IF VAT.bAbisoliererLINKSundAUF AND NOT VAT.bNurAbisolieren THEN
	VAT.bAbisoliererLINKSundAUF := FALSE;
	VAT.bCrimpeinheitVOR := TRUE; //M20.4
	GVL.EinzelschrittIdx := einzelSchrittOffset + 25; //NBT-NEU: Crimpeinheit vor
	MAIN.M_Log(reqLevel:=CVL.TRACE, objectName:= 'Ablauf', sMsg:= '4---Crimper vor',errNo := 16#FFFFFFFF);
	RETURN;
END_IF

(*	
	//*** 5---Crimpen zu
	U "M 20.4" M20.4 -- 4---Crimpeinheit vor
	R "M 20.4" M20.4 -- 4---Crimpeinheit vor
	S "M 20.5" M20.5 -- 5---Crimpen zu
	R "M 23.3" M23.3 -- S&R 2ter Vereinzelungs-Versuch
	SPB end
*)
	
IF VAT.bCrimpeinheitVOR THEN //M20.4
	VAT.bCrimpeinheitVOR := FALSE; //M20.4
	VAT.bCrimpenZU := TRUE; //M20.5
	VAT.bSr2terVereinzVersuch := FALSE; //M23.3
	GVL.EinzelschrittIdx := einzelSchrittOffset + 26; //NBT-NEU: Crimpen zu
	MAIN.M_Log(reqLevel:=CVL.TRACE, objectName:= 'Ablauf', sMsg:= '5---Crimper zu',errNo := 16#FFFFFFFF);
	RETURN;
END_IF
	
(*	
	//*** 6---Drahthalter + Drahtführung auf
	U "M 20.5" M20.5 -- 5---Crimpen zu
	R "M 20.5" M20.5 -- 5---Crimpen zu
	S "M 20.6" M20.6 -- 6---Drahthalter + Drahtführung auf
	SPB end
*)
	
IF VAT.bCrimpenZU THEN //Crimpen zu
	VAT.bCrimpenZU := FALSE;
	VAT.bDrahtHalterUndFuehrungAUF := TRUE;
	GVL.EinzelschrittIdx := einzelSchrittOffset + 27; //NBT-NEU: Drahthalter + Drahtführung auf
	MAIN.M_Log(reqLevel:=CVL.TRACE, objectName:= 'Ablauf', sMsg:= '6---Draht auf',errNo := 16#FFFFFFFF);
	RETURN;
END_IF
	
(*		
	//*** 7---Crimpzange auf + Abisoliereinheit vor
	U "M 20.6" M20.6 -- 6---Drahthalter + Drahtführung auf
	R "M 20.6" M20.6 -- 6---Drahthalter + Drahtführung auf
	S "M 20.7" M20.7 -- 7---Crimpzange auf + Abisoliereinheit vor
	SPB end
*)
		
IF VAT.bDrahtHalterUndFuehrungAUF THEN //Drahthalter + Drahtführung auf
	VAT.bDrahtHalterUndFuehrungAUF := FALSE; //M20.6
	VAT.bCrZangeAUF_AisolierVOR := TRUE; //M20.7
	GVL.EinzelschrittIdx := einzelSchrittOffset + 28; //NBT-NEU: Crimpzange auf + Abisoliereinheit vor
	MAIN.M_Log(reqLevel:=CVL.TRACE, objectName:= 'Ablauf', sMsg:= '7---C-Zange auf, AbIso vor',errNo := 16#FFFFFFFF);
	RETURN;
END_IF

(*		
	//*** 8---Ausstoßen vor
	L "DB6".w134_Ausstossverz DB6.DBW134 -- Ausstoß-Verzögerung
	L 10
	*I -- AKKU1 und AKKU2 multiplizieren, Das Ergebnis wird in AKKU 1 abgelegt.
	ITB -- Ganzzahl in BCD umwandeln (3 Stellen und eine Stelle Vorzeichen)
	
	U "M 20.7" M20.7 -- 7---Crimpzange auf + Abisoliereinheit vor
	SE "T 22" T22 -- Ausstoß-Verzögerung
	U "T 22" T22 -- Ausstoß-Verzögerung
	R "M 20.7" M20.7 -- 7 Crimpzange auf + Abisoliereinheit vor
	S "M 21.0" M21.0 -- 8---Ausstoßen vor
	SPB end
*)

//ITB ??? Wert befindet sich in AKKU 1, wird aber nicht weggeschrieben...was passiert damit?
//nach vorn verlagert
//GVL.tonAusstoss(IN := VAT.bCrZangeAUF_AisolierVOR, PT := INT_TO_TIME (nTmp)); 

IF GVL.tonAusstoss.Q THEN
	VAT.bCrZangeAUF_AisolierVOR := FALSE; //M20.7
	VAT.bAusstossenVOR := TRUE; //M21.0
	GVL.EinzelschrittIdx := einzelSchrittOffset + 29; //NBT-NEU: Ausstoßen vor
	MAIN.M_Log(reqLevel:=CVL.TRACE, objectName:= 'Ablauf', sMsg:= '8---Ausstoßen vor',errNo := 16#FFFFFFFF);
	RETURN;
ELSE	
	GVL.EinzelschrittIdx := einzelSchrittOffset + 29; //NBT-NEU: Ausstoßen vor
END_IF

(*		
	//*** 9---Crimpeinheit rück
	U "M 21.0" M21.0 -- 8---Ausstoßen vor
	R "M 21.0" M21.0 -- 8---Ausstoßen vor
	S "M 21.1" M21.1 -- 9---Crimpeinheit rück
	SPB end
*)
	
IF VAT.bAusstossenVOR THEN //M21.0
	VAT.bAusstossenVOR := FALSE;
	VAT.bCrimpeinheitRUECK := TRUE; //M21.1
	GVL.EinzelschrittIdx := einzelSchrittOffset + 30; //NBT-NEU: Crimpeinheit rück
	MAIN.M_Log(reqLevel:=CVL.TRACE, objectName:= 'Ablauf', sMsg:= '9---Crimper rück',errNo := 16#FFFFFFFF);
	RETURN;
END_IF
(*		
	//*** 10--Abisolierer nach rechts + Kontakt-Schieben rück
	U "M 20.3" M20.3 -- 3---Abisolierer nach links + Abisolierer auf
	U "M8.4NurAbisolieren" M8.4 -- Nur Abisolieren
	UN "T 20" T20 -- Ablauf-Verz.bei Probelauf
	O "M 21.1" M21.1 -- 9---Crimpeinheit rück
	SPBN l10
*)
	
//SPBN -> Springe wenn VKE = 0 -> 'Springe bei FALSE' heißt 'Tu was bei TRUE'.
IF VAT.bAbisoliererLINKSundAUF AND VAT.bNurAbisolieren AND NOT GVL.tofAblVerzProbelauf.Q OR VAT.bCrimpeinheitRUECK THEN
	
	MAIN.M_Log(reqLevel:=CVL.TRACE, objectName:= 'Ablauf', sMsg:= '10--Abisolierer re + K-Schieber rück',errNo := 16#FFFFFFFF);
	(*	
		R "M 20.3" M20.3 -- 3---Abisolierer nach links + Abisolierer auf
		R "M 21.1" M21.1 -- 9---Crimpeinheit rück
		S "M 21.2" M21.2 -- 10--Abisolierer nach rechts + Kontakt-Schieben rück
	*)
	VAT.bAbisoliererLINKSundAUF := FALSE; //M20.3
	VAT.bCrimpeinheitRUECK := FALSE; //M21.1
	VAT.bAbisoNachRE_KontSchiebRUECK := TRUE; //M21.2

	(*	
		U "M8.7ohneLitze" M8.7 -- Probelauf ohne Litze
		R "M8.7ohneLitze" M8.7 -- Probelauf ohne Litze
		R "M0.6" M0.6 -- SR Start
	*)
	
	IF VAT.bProbelOhneLitze THEN // Probelauf ohne Litze //M8.7
		VAT.bProbelOhneLitze := FALSE; //M8.7
		VAT.bSrStart := FALSE; //SR Start - M0.6
	END_IF
	
	(*	
		O "M8.5ohneKontakt" M8.5 -- Probelauf ohne Kontakt
		O "M8.6ohneCrmpen" M8.6 -- Probelauf ohne Crimpen
		L S5T#600MS
		SA "T 20" T20 -- Ablauf-Verz.bei Probelauf
		CLR
		SA "T 20" T20 -- Ablauf-Verz.bei Probelauf
	*)
	

	GVL.tofAblVerzProbelauf(IN := VAT.bProbelOhneKontakt OR VAT.bProbelOhneCrimpen, PT := T#600MS); //T20
	
	(*
		U "M8.0NormalCrimp" M8.0 -- Normal Crimpen
		SPBN l10
	*)
	
	//SPBN -> Springe wenn VKE = 0 -> 'Springe bei FALSE' heißt 'Tu was bei TRUE'.
	IF VAT.bNormalCrimp THEN // Normal Crimpen
		(*	
			L "DB6".d140_Total_Z DB6.DBD140 -- Total-Zähler
			+ L#1
			T "DB6".d140_Total_Z DB6.DBD140 -- Total-Zähler
			L "DB6".d144_Tages_Z DB6.DBD144 -- Tages-Zähler
			+ L#1
			T "DB6".d144_Tages_Z DB6.DBD144 -- Tages-Zähler
			L "DB6".d68Stueck_Fertig DB6.DBD68 -- Fertig Stückz
			+ L#1
			T "DB6".d68Stueck_Fertig DB6.DBD68 -- Fertig Stückz
			L "DB6".d64Stueck_Vorwahl DB6.DBD64 -- Stückzahl-Vorwahl Stückz
			==D
			S "A70" M107.0 -- Stückzahl-Vorwahl erreicht
			
			L "DB6".d152_WartZ_Z DB6.DBD152 -- Zähler Wartung
			+ L#1
			T "DB6".d152_WartZ_Z DB6.DBD152 -- Zähler Wartung
			
			L "DB6".d148_WartZ_V DB6.DBD148 -- Vorwahl Wartung
			==D
			S "A67" M106.7 -- Wartungs-Zähler, hat Vorwahl erreicht, weiter mit Reset
			SPA end
		*)
					
		
		DB6.diTotalZaehler := DB6.diTotalZaehler + 1;
		
		DB6.diTagesZaehler := DB6.diTagesZaehler + 1;
					
		DB6.diStueck_Fertig := DB6.diStueck_Fertig + 1;
		
		IF DB6.diStueck_Fertig = DB6.diStueck_Vorwahl THEN
			GVL.errs.StueckZaehlErreicht := TRUE; //M107.0
		END_IF
		
		
		DB6.diWartungsZaehler := DB6.diWartungsZaehler + 1;
		
		IF DB6.diWartungsZaehler = DB6.diWartZaehlVorwahl THEN
			GVL.errs.WartungsZaehlErreicht := TRUE; //M106.7
			GVL.EinzelschrittIdx := einzelSchrittOffset + 31; //NBT-NEU: Abisolierer nach rechts + Kontakt-Schieben rück
			RETURN; //Wartungs-Zähler, hat Vorwahl erreicht, weiter mit Reset
		END_IF

	END_IF // end of IF VAT.M8.0...

END_IF //end of IF VAT.M20.3 AND VAT.M8.4 AND NOT ...

(*	
l10: BLD 130
	U "M 21.2" M21.2 -- 10--Abisolierer nach rechts + Kontakt-Schieben rück
	R "M 21.2" M21.2 -- 10--Abisolierer nach rechts + Kontakt-Schieben rück
*)

IF VAT.bAbisoNachRE_KontSchiebRUECK THEN //M21.2
	VAT.bAbisoNachRE_KontSchiebRUECK := FALSE; //M21.2
	GVL.EinzelschrittIdx := einzelSchrittOffset + 32; // Einzelschritt Ende
	MAIN.M_Log(reqLevel:=CVL.TRACE, objectName:= 'Ablauf', sMsg:= '10--ENDE',errNo := 16#FFFFFFFF);
END_IF

(*	
end: BLD 130
*)

END_FUNCTION_BLOCK

// ---- POUs/MainPous/F20_Ablauf/P_AblaufReset.TcPOU
PROGRAM P_AblaufReset 
VAR
//rTrig : R_TRIG;
//bTmp:BOOL := FALSE;
tsv1 : TSV;	

END_VAR

(* Netzwerk: 2 Ablauf-Reset *)

(* 
U "E0_0" E0.0	-- Taste Start
U "M0.7" M0.7	-- Störung aufgetreten (gesammelt)
L S5T#1S		-- mandatory!
SE "T 1" T1 -- Verz. Taste Start, SE <Zeit> startet die adressierte Zeit, wenn das VKE von "0" auf "1" wechselt.
*)

(*
Klassisches TON-Verhalten:
Die programmierte Zeitdauer läuft ab, solange das VKE = 1 ist. Wechselt das VKE auf "0", bevor die programmierte
Zeitdauer abgelaufen ist, wird die Zeit angehalten. Für diese Operation (Starten der Zeit) müssen der
Zeitwert und die Zeitbasis im BCD-Format in AKKU1-L gespeichert sein.
*)
//Also nur wenn eine Sammelstörung aufgetreten ist und 1 sek. gedrückt wird!...
GVL.tonTasteStartOnErr(IN := GVL.insecTasterStart AND VAT.bSammelStoerung, PT := T#1S);

(*
	ON "T 72" T72 -- Verz. Alles OK von PNOZ
	O "T 1" T1 -- Verz. Taste Start
	SPBN res -- Springe nach 'res' wenn VKE = 0

	R "M8.1MagLeerf" M8.1 -- Magazin Leerfahren
	R "M8.2SortLeerf" M8.2 -- Sortierer Leerfahren
	R "M8.3CrimpEinr" M8.3 -- Crimpen Einrichten
	R "M8.5ohneKontakt" M8.5 -- Probelauf ohne Kontakt
	R "M8.6ohneCrmpen" M8.6 -- Probelauf ohne Crimpen
	R "M8.7ohneLitze" M8.7 -- Probelauf ohne Litze

	L 0
	T MD 20 -- Bedeutung noch Unklar
	T MW 0 -- Bedeutung noch Unklar
	T AW 0 -- Bedeutung noch Unklar
	T AW 2 -- Bedeutung noch Unklar
	T MD 104 -- Bedeutung noch Unklar
	T MD 108 -- Bedeutung noch Unklar
	SET -- 	VKE auf 1 setzen (=1)
	S "M1.3_Stop" M1.3 -- RS Stop StST
*)

IF (* NOT GVL.tonSAFETYok.Q OR *) GVL.tonTasteStartOnErr.Q THEN
	VAT.bMagazinLeerfahren := FALSE;
	VAT.bSortiererLeerfahren := FALSE;
	VAT.bCrimpEinrichten := FALSE;
	VAT.bProbelOhneKontakt := FALSE;
	VAT.bProbelOhneCrimpen := FALSE;
	VAT.bProbelOhneLitze := FALSE;
	
	//GVL.MD20 := 0; //Bedeutung noch Unklar
	//GVL.MW0 := 0; //Bedeutung noch Unklar
	//T AW 0 -- Bedeutung noch Unklar(evtl. alle 8 Ausg. auf 0)
	//T AW 2 -- Bedeutung noch Unklar (evtl. alle 8 Ausg. als WORD auf 2)
	//GVL.MD104 := 0; //war Fehererkennung, jtzt GVL.errs
	//GVL.MD108 := 0; //war Fehererkennung, jtzt GVL.errs
	
	F_ResetErrors(); //Reset Fehlerflags
	
	VAT.bRsStop := TRUE; //(ehemals M1.3) RS Stop
END_IF

(*	
res: BLD 130
	U "T 72" T72 -- Verz. Alles OK von PNOZ
	L S5T#500MS
	SV "T 19" T19 -- Kontaktauswurf nach Einschalten, Zeit als Zeit mit verlängertem Impuls starten: TSV.
*)

GVL.tsvKontauswurf(IN := GVL.tonSAFETYok.Q, PT := T#500MS);

END_PROGRAM

// ---- POUs/MainPous/FC3_FehlerAllg/F_ResetErrors.TcPOU
FUNCTION F_ResetErrors : BOOL
VAR_INPUT
END_VAR
VAR
END_VAR

//M104.0
	GVL.errs.DrahthltNichtOffen := FALSE; //(ehem. M104.0) Drahthalter nicht offen
	GVL.errs.DrahthltNichtZu := FALSE; //(ehem. M104.1) Drahthalter nicht zu
	GVL.errs.AusloesSchaltDauerMldg := FALSE;//(ehem. M104.2) -- Auslöseschalter Dauermelung
	GVL.errs.AbisolierNichtOffen  := FALSE; //(ehem. M104.3) Abisolierer nicht offen
	GVL.errs.AbisolierNichtZu  := FALSE; //(ehem. M104.4) Abisolierer nicht zu
	GVL.errs.DoppelMlgAbisoVornRueck  := FALSE; //(ehem. M104.5) Doppelmeldung Abisolierer vorn+rück
	GVL.errs.AbisolierNichtVorn  := FALSE; //(ehem. M104.6) Abisolierer nicht vorn
	GVL.errs.AbisolierNichtRueck  := FALSE; //(ehem. M104.7) Abisolierer nicht rück (abisoliert)
	
	//M105.0
	GVL.errs.AbisolierNichtLinks  := FALSE; //(ehem. M105.0) Abisolierer nicht links (aus Arbeitsraum)
	GVL.errs.AbisolierNichtRechts  := FALSE; //(ehem. M105.1) Abisolierer nicht rechts
	GVL.errs.DoppelMlgCrimpzZuOffen  := FALSE; //(ehem. M105.2) Doppelmeldung Crimpzange zu+offen
	GVL.errs.CrimpZangeNichtZu  := FALSE; //(ehem. M105.3) Crimpzange nicht zu
	GVL.errs.CrimpZangeNichtOffen  := FALSE; //(ehem. M105.4) Crimpzange nicht offen
	GVL.errs.KontaktNichtGefallen  := FALSE; //Reserve, war in AWL nicht belegt
	GVL.errs.DauerMlgKontaktGefallen  := FALSE; //Reserve, war in AWL nicht belegt
	GVL.errs.DoppelMlgCrimpEinhVornZurueck  := FALSE; //(ehem. M105.7) Doppelmeldung Crimpeinheit vorn+rück
	
	//M106.0
	GVL.errs.CrimpeinheitNichtVorn  := FALSE; //(ehem. M106.0)Crimpeinheit nicht vorn
	GVL.errs.CrimpeinheitNichtRueck  := FALSE; //(ehem. M106.1) Crimpeinheit nicht rück
	GVL.errs.KontaktSchiebenNichtVorn  := FALSE; //(ehem. M106.2) Kontakt-Schieben nicht vorn
	GVL.errs.KontaktSchiebenNichtRueck  := FALSE; //(ehem. M106.3) Kontakt-Schieben nicht rück
	GVL.errs.AusstossenNichtVorn  := FALSE; //(ehem. M106.4) Ausstoßen nicht vorn
	GVL.errs.AusstossenNichtRueck  := FALSE; //(ehem. M106.5) Ausstoßen nicht rück
	GVL.errs.r106_6  := FALSE; //Reserve, war in AWL nicht belegt
	GVL.errs.WartungsZaehlErreicht := FALSE; //(ehem. M106.7) Wartungs-Zähler, hat Vorwahl erreicht
	
	//M107.0
	GVL.errs.StueckZaehlErreicht := FALSE; //(ehem. M107.0 Stückzahl-Vorwahl erreicht)
	GVL.errs.r107_1  := FALSE; //Reserve, war in AWL nicht belegt
	GVL.errs.r107_2  := FALSE; //Reserve, war in AWL nicht belegt
	GVL.errs.r107_3  := FALSE; //Reserve, war in AWL nicht belegt
	GVL.errs.r107_4  := FALSE; //Reserve, war in AWL nicht belegt
	GVL.errs.r107_5  := FALSE; //Reserve, war in AWL nicht belegt
	GVL.errs.r107_6  := FALSE; //Reserve, war in AWL nicht belegt
	GVL.errs.r107_7  := FALSE; //Reserve, war in AWL nicht belegt

END_FUNCTION

// ---- POUs/MainPous/F20_Ablauf/F_AblaufketteLeerfahren.TcPOU
FUNCTION F_AblaufketteLeerfahren : BOOL
VAR_INPUT
END_VAR
VAR
	
END_VAR

(* Netzwerk: 4 Ablaufkette Leerfahren oder Cripen einrichten *)

//Timer muss immer durchlaufen werden. TOF kann permanent auf FALSE gelassen werden, wenn er eine Start-Flanke erhalten hat.
GVL.tofMagazLeerFahr(IN := FALSE, PT := T#500MS);


(*
	U "M 22.7" M22.7 -- Endstellung
	SPBN l0
*)

//SPBN -> Springe wenn VKE = 0 -> 'Springe bei FALSE' heißt 'Tu was bei TRUE'.
IF VAT.bEndstellung THEN

	(*	
		O "M8.1MagLeerf" M8.1 -- Magazin Leerfahren
		O "M8.2SortLeerf" M8.2 -- Sortierer Leerfahren
		O "M8.3CrimpEinr" M8.3 -- Crimpen Einrichten
		U "M 3.0" M3.0 -- Alles in Sollposition
		SPBN l0
		
		S "M 22.0" M22.0 -- 0---Abisolierer nach Links Leerf-o-Ce -- S (Setze Bit) schreibt bei VKE = 1 (und MCR = 1) den Wert "1" in das adressierte Bit.
		SPB Lend
	*)

	//SPBN -> Springe wenn VKE = 0 -> 'Springe bei FALSE' heißt 'Tu was bei TRUE'.
	IF (VAT.bMagazinLeerfahren OR VAT.bSortiererLeerfahren OR VAT.bCrimpEinrichten) AND VAT.bAllesInSollPos THEN

		//'Statemachine' Start:
		VAT.bAbisoliererNachLinksLoC := TRUE; //wenn er nicht gesprungen ist, muss VKE 1 gewesen sein, dehalb stumpf TRUE.
		RETURN;
		
	END_IF
END_IF
		
(*
l0: BLD 130

	//*** 1---Crimpeinheit vor Leerf-ohne-Ce
	U "M 22.0" M22.0 -- 0---Abisolierer nach Links Leerf-o-Ce
	U "M 3.0" M3.0 -- Alles in Sollposition
	R "M 22.0" M22.0 -- 0---Abisolierer nach Links Leerf-o-Ce
	S "M 22.1" M22.1 -- 1---Crimpeinheit vor Leerf-o-Ce
	SPB Lend
*)
	
IF VAT.bAbisoliererNachLinksLoC AND VAT.bAllesInSollPos THEN
	VAT.bAbisoliererNachLinksLoC := FALSE;	//M22.0
	VAT.bCrimpEinheitVorLoC := TRUE; //M22.1
	RETURN;
END_IF
	
(*	
	//*** 2---Vereinzelung takten od. Crimpen zu/auf Leerf-o-Ce
	U "M 22.1" M22.1 -- 1---Crimpeinheit vor Leerf-o-Ce
	U "M 3.0" M3.0 -- Alles in Sollposition
	R "M 22.1" M22.1 -- 1---Crimpeinheit vor Leerf-o-Ce
	S "M 22.2" M22.2 -- 2---Vereinzelung takten od.Crimpen zu/auf Leerf-o-Ce
	SPB Lend
*)	
	
IF VAT.bCrimpEinheitVorLoC AND VAT.bAllesInSollPos THEN
	VAT.bCrimpEinheitVorLoC := FALSE;	 //M22.1
	VAT.bVereinzelungTakten := TRUE; //M22.2
	RETURN;
END_IF
	
(*	
	U "M 22.2" M22.2 -- 2---Vereinzelung takten od.Crimpen zu/auf Leerf-o-Ce
	SPBN l3
*)

//SPBN -> Springe wenn VKE = 0 -> 'Springe bei FALSE' heißt 'Tu was bei TRUE'.
IF VAT.bVereinzelungTakten THEN
	(*	
		U "M8.3CrimpEinr" M8.3 -- Crimpen Einrichten
		U "M 80.0" M80.0 -- +F E0.0 Taste Start
		SPBN caz
	*)
	
	IF VAT.bCrimpEinrichten AND VAT.bFlkTasteStart THEN
		(*	
		UN "M 22.6" M22.6 -- Crimpen zu bei Einstellen Leerf-o-Ce
		= "M 22.6" M22.6 -- Crimpen zu bei Einstellen Leerf-o-Ce
		*)
		VAT.bCrimpenZuBeiEinstellen := NOT VAT.bCrimpenZuBeiEinstellen;	 //M22.6
	END_IF 
	
	(*		
	caz: O "M8.1MagLeerf" M8.1 -- Magazin Leerfahren
		O "M8.2SortLeerf" M8.2 -- Sortierer Leerfahren
		UN "T 41" T41 -- Takt für Magazin leerfahren
		SPBN kl
		
		L S5T#500MS
		SA "T 41" T41 -- Takt für Magazin leerfahren
		CLR
		SA "T 41" T41 -- Takt für Magazin leerfahren
		UN "M 23.0" M23.0 -- Takt für Vereinzelung bei Leerfahren
		= "M 23.0" M23.0 -- Takt für Vereinzelung bei Leerfahren
		//*** 3---Crimpeinheit rück Leerf-o-Ce
	*)
	IF (VAT.bMagazinLeerfahren OR VAT.bSortiererLeerfahren) AND NOT GVL.tofMagazLeerFahr.Q THEN
		GVL.tofMagazLeerFahr(IN := TRUE, PT := T#500MS);
		VAT.bTaktVereinzLeerF := NOT VAT.bTaktVereinzLeerF;	
	END_IF
	
	(*	
	kl: UN "M8.1MagLeerf" M8.1 -- Magazin Leerfahren
		UN "M8.2SortLeerf" M8.2 -- Sortierer Leerfahren
		UN "M8.3CrimpEinr" M8.3 -- Crimpen Einrichten
		UN "M 23.0" M23.0 -- Takt für Vereinzelung bei Leerfahren
		R "M 22.2" M22.2 -- 2---Vereinzelung takten od.Crimpen zu/auf Leerf-o-Ce
		S "M 22.3" M22.3 -- 3---Crimpeinheit rück Leerf-o-Ce
		R "M 22.6" M22.6 -- Crimpen zu bei Einstellen Leerf-o-Ce
		SPB Lend
	*)	
	
	IF NOT VAT.bMagazinLeerfahren AND NOT VAT.bSortiererLeerfahren AND NOT VAT.bCrimpEinrichten  AND NOT VAT.bTaktVereinzLeerF THEN
		VAT.bVereinzelungTakten := FALSE;
		VAT.bCrimpEinheitRueckLoC := TRUE;
		VAT.bCrimpenZuBeiEinstellen := FALSE;
		RETURN;
	END_IF //end of IF VAT.M22.2
		
END_IF // end of IF VAT.bVereinzelungTakten

(*	
l3: BLD 130
	U "M 22.3" M22.3 -- 3---Crimpeinheit rück Leerf-o-Ce
	U "M 3.0" M3.0 -- Alles in Sollposition
	R "M 22.3" M22.3 -- 3---Crimpeinheit rück Leerf-o-Ce
*)

IF VAT.bCrimpEinheitRueckLoC AND VAT.bAllesInSollPos THEN
	VAT.bCrimpEinheitRueckLoC := FALSE; //M22.3
END_IF
	
(*	
Lend: BLD 130
*)

END_FUNCTION

// ---- POUs/MainPous/F20_Ablauf/F_Endstellung.TcPOU
FUNCTION F_Endstellung : BOOL
VAR_INPUT
END_VAR
VAR
END_VAR

(* Netzwerk: 5 Endstellung *)

(*
UN "M 20.0" M20.0 -- 0---Drahthalter + Drahtführung zu
UN "M 20.1" M20.1 -- 1---Abisolierer zu
UN "M 20.2" M20.2 -- 2---Abisolierer rück (abisolieren)
UN "M 20.3" M20.3 -- 3---Abisolierer nach links + Abisolierer auf
UN "M 20.4" M20.4 -- 4---Crimpeinheit vor
UN "M 20.5" M20.5 -- 5---Crimpen zu
UN "M 20.6" M20.6 -- 6---Drahthalter + Drahtführung auf
UN "M 20.7" M20.7 -- 7---Crimpzange auf + Abisoliereinheit vor

UN "M 21.0" M21.0 -- 8---Ausstoßen vor
UN "M 21.1" M21.1 -- 9---Crimpeinheit rück
UN "M 21.2" M21.2 -- 10--Abisolierer nach rechts + Kontakt-Schieben rück

UN "M 22.0" M22.0 -- 0---Abisolierer nach Links Leerf-o-Ce
UN "M 22.1" M22.1 -- 1---Crimpeinheit vor Leerf-o-Ce
UN "M 22.2" M22.2 -- 2---Vereinzelung takten od.Crimpen zu/auf Leerf-o-Ce
UN "M 22.3" M22.3 -- 3---Crimpeinheit rück Leerf-o-Ce

= "M 22.7" M22.7 -- Endstellung

*)

VAT.bEndstellung := 
	//M20.X
	NOT VAT.bDrahtHalterUndFuehrungZU AND
	NOT VAT.bAbisoliererZU AND
	NOT VAT.bAbisoliererRUECK AND
	NOT VAT.bAbisoliererLINKSundAUF AND
	NOT VAT.bCrimpeinheitVOR AND
	NOT VAT.bCrimpenZU AND
	NOT VAT.bDrahtHalterUndFuehrungAUF AND
	NOT VAT.bCrZangeAUF_AisolierVOR AND
	//M21.X
	NOT VAT.bAusstossenVOR AND
	NOT VAT.bCrimpeinheitRUECK AND
	NOT VAT.bAbisoNachRE_KontSchiebRUECK AND
	//M22.X
	NOT VAT.bAbisoliererNachLinksLoC AND
	NOT VAT.bCrimpEinheitVorLoC AND
	NOT VAT.bVereinzelungTakten AND
	NOT VAT.bCrimpEinheitRueckLoC;
	
F_Endstellung := VAT.bEndstellung;

END_FUNCTION

// ---- POUs/MainPous/F20_Ablauf/F_Ventile.TcPOU
FUNCTION F_Ventile : BOOL
VAR_INPUT
END_VAR
VAR
	wDrahthalterSchliessdruck : UINT := 0;
END_VAR

(* Netzwerk: 6 Ventile *)

	(*
	U "E1_7" E1.7 -- R Crimpzange offen
	L S5T#50MS
	SA "T 31" T31 -- Verl. E1.7 Crimpzange offen
	*)
	
	GVL.tofCrimpzangeOffen(IN := GVL.insecCrimpZangeIstOFFEN, PT := T#50MS);
	
	(*
	U "M 20.3" M20.3 -- 3---Abisolierer nach links + Abisolierer auf
	UN "M8.4NurAbisolieren" M8.4 -- Nur Abisolieren
	O "M 20.0" M20.0 -- 0---Drahthalter + Drahtführung zu
	O "M 20.1" M20.1 -- 1---Abisolierer zu
	O "M 20.2" M20.2 -- 2---Abisolierer rück (abisolieren)
	O "M 20.4" M20.4 -- 4---Crimpeinheit vor
	O(
	U "M 20.5" M20.5 -- 5---Crimpen zu
	U "T 31" T31 -- Verl. E1.7 Crimpzange offen
	)
	= "A 1.7" A1.7 -- Y-10 Drahthalter+Führung zu
	*)
	
	IO.outY10DrahthaltFuehrungZU := 
		(VAT.bAbisoliererLINKSundAUF AND
		NOT VAT.bNurAbisolieren) OR
		VAT.bDrahtHalterUndFuehrungZU OR
		VAT.bAbisoliererZU OR
		VAT.bAbisoliererRUECK OR
		VAT.bCrimpeinheitVOR OR
		(VAT.bCrimpenZU AND GVL.tofCrimpzangeOffen.Q);

	(*
	L 0  -- im VKE steht noch A1.7 ...
	SPBN dr
	*)
	
	IF IO.outY10DrahthaltFuehrungZU THEN 
		(*
		L "DB6".d376 DB6.DBD376
		L 2.730000e+003 //Faktor 6*2730=3FFF (10V)
		*R
		RND -- Gleitpunktzahl zur Ganzzahl runden
		*)
		//ToDo: Testen: 4-20mA diese originale Linearisierung nehmen oder PArametrierung erlauben?
		wDrahthalterSchliessdruck := REAL_TO_UINT(DB6.rDrahthalterSchliessdruck * 2.730000E+003);
	ELSE
		wDrahthalterSchliessdruck := 0;
	END_IF
(*
dr: T "AW 6" AW6 -- Drahthalter Schließdruck
*)
	IO.outSollwertDruckVentil := wDrahthalterSchliessdruck;

	(*
	O "M 20.2" M20.2 -- 2---Abisolierer rück (abisolieren)
	O "M 20.3" M20.3 -- 3---Abisolierer nach links + Abisolierer auf
	= "A 1.5" A1.5 -- Y-8 Abisolierer rück
	*)
	IO.outY8AbisoliererRUECK := VAT.bAbisoliererRUECK OR VAT.bAbisoliererLINKSundAUF;
	
	(*
	O "M 20.1" M20.1 -- 1---Abisolierer zu
	O "M 20.2" M20.2 -- 2---Abisolierer rück (abisolieren)
	O "M 20.4" M20.4 -- 4---Crimpeinheit vor
	O "M 20.5" M20.5 -- 5---Crimpen zu
	O "M 20.6" M20.6 -- 6---Drahthalter + Drahtführung auf
	O "M 20.7" M20.7 -- 7---Crimpzange auf + Abisoliereinheit vor
	O "M 21.0" M21.0 -- 8---Ausstoßen vor
	O "M 21.1" M21.1 -- 9---Crimpeinheit rück
	O "M 22.0" M22.0 -- 0---Abisolierer nach LinksLeerf-o-Ce
	O "M 22.1" M22.1 -- 1---Crimpeinheit vorLeerf-o-Ce
	O "M 22.2" M22.2 -- 2---Vereinzelung takten od.Crimpen zu/auf Leerf-o-Ce
	O "M 22.3" M22.3 -- 3---Crimpeinheit rückLeerf-o-Ce
	= "A 1.3" A1.3 -- Y-6 Abisolierer zu
	*)
	IO.outY6AbisoliererZU :=	VAT.bAbisoliererZU OR //Abisolierer zu
							VAT.bAbisoliererRUECK OR //Abisolierer rück (abisolieren)
							VAT.bCrimpeinheitVOR OR //Crimpeinheit vor
							VAT.bCrimpenZU OR //Crimpen zu
							VAT.bDrahtHalterUndFuehrungAUF OR //Drahthalter + Drahtführung auf
							VAT.bCrZangeAUF_AisolierVOR OR //Crimpzange auf + Abisoliereinheit vor
							VAT.bAusstossenVOR OR //Ausstoßen vor
							VAT.bCrimpeinheitRUECK OR //Crimpeinheit rück
							VAT.bAbisoliererNachLinksLoC OR //Abisolierer nach LinksLeerf-o-Ce
							VAT.bCrimpEinheitVorLoC OR //Crimpeinheit vorLeerf-o-Ce
							VAT.bVereinzelungTakten OR //Vereinzelung takten od.Crimpen zu/auf Leerf-o-Ce
							VAT.bCrimpEinheitRueckLoC ;  //Crimpeinheit rückLeerf-o-Ce
	(*
	O "M 20.3" M20.3 -- 3---Abisolierer nach links + Abisolierer auf
	O "M 20.4" M20.4 -- 4---Crimpeinheit vor
	O "M 20.5" M20.5 -- 5---Crimpen zu
	O "M 20.6" M20.6 -- 6---Drahthalter + Drahtführung auf
	O "M 20.7" M20.7 -- 7---Crimpzange auf + Abisoliereinheitvor
	O "M 21.0" M21.0 -- 8---Ausstoßen vor
	O "M 21.1" M21.1 -- 9---Crimpeinheit rück
	O "M 22.0" M22.0 -- 0---Abisolierer nach LinksLeerf-o-Ce
	O "M 22.1" M22.1 -- 1---Crimpeinheit vorLeerf-o-Ce
	O "M 22.2" M22.2 -- 2---Vereinzelung takten od.Crimpen zu/auf Leerf-o-Ce
	O "M 22.3" M22.3 -- 3---Crimpeinheit rückLeerf-o-Ce
	= "A 1.2" A1.2 -- Y-5 Abisolierer nach links+Abdeckungzu
	= "A 1.4" A1.4 -- Y-7 Abfall runter
	*)
	IO.outY5AbisolierNachLINKS :=	VAT.bAbisoliererLINKSundAUF OR // Abisolierer nach links + Abisolierer auf
								VAT.bCrimpeinheitVOR OR // Crimpeinheit vor
								VAT.bCrimpenZU OR // Crimpen zu
								VAT.bDrahtHalterUndFuehrungAUF OR // Drahthalter + Drahtführung auf
								VAT.bCrZangeAUF_AisolierVOR OR // Crimpzange auf + Abisoliereinheitvor
								VAT.bAusstossenVOR OR // Ausstoßen vor
								VAT.bCrimpeinheitRUECK OR // Crimpeinheit rück
								VAT.bAbisoliererNachLinksLoC OR // Abisolierer nach LinksLeerf-o-Ce
								VAT.bCrimpEinheitVorLoC OR // Crimpeinheit vorLeerf-o-Ce
								VAT.bVereinzelungTakten OR // Vereinzelung takten od.Crimpen zu/auf Leerf-o-Ce
								VAT.bCrimpEinheitRueckLoC ;  // Crimpeinheit rückLeerf-o-Ce
	
	IO.outY7AbfallRUNTER := IO.outY5AbisolierNachLINKS;							

	(*
	O "M 20.4" M20.4 -- 4---Crimpeinheit vor
	O "M 20.5" M20.5 -- 5---Crimpen zu
	O "M 20.6" M20.6 -- 6---Drahthalter + Drahtführung auf
	O "M 20.7" M20.7 -- 7---Crimpzange auf + Abisoliereinheitvor
	O "M 21.0" M21.0 -- 8---Ausstoßen vor
	O "M 22.1" M22.1 -- 1---Crimpeinheit vor Leerf-o-Ce
	O "M 22.2" M22.2 -- 2---Vereinzelung takten od.Crimpen zu /auf Leerf-o-Ce
	= "A 1.1" A1.1 -- Y-4 Crimpeinheit vor
	*)
	
	IO.outY4CrimpEinheitVOR :=	VAT.bCrimpeinheitVOR OR // Crimpeinheit vor
								VAT.bCrimpenZU OR // Crimpen zu
								VAT.bDrahtHalterUndFuehrungAUF OR // Drahthalter + Drahtführung auf
								VAT.bCrZangeAUF_AisolierVOR OR // Crimpzange auf + Abisoliereinheitvor
								VAT.bAusstossenVOR OR // Ausstoßen vor
								VAT.bCrimpEinheitVorLoC OR // Crimpeinheit vorLeerf-o-Ce
								VAT.bVereinzelungTakten ;  // Vereinzelung takten od.Crimpen zu/auf Leerf-o-Ce
								
	
	(*
	O "M 20.3" M20.3 -- 3---Abisolierer nach links + Abisolierer auf
	O "M 20.4" M20.4 -- 4---Crimpeinheit vor
	O "M 20.5" M20.5 -- 5---Crimpen zu
	O "M 20.6" M20.6 -- 6---Drahthalter + Drahtführung auf
	O "M 20.7" M20.7 -- 7---Crimpzange auf + Abisoliereinheitvor
	O "M 21.0" M21.0 -- 8---Ausstoßen vor
	O "M 21.1" M21.1 -- 9---Crimpeinheit rück
	O "T 19" T19 -- Kontaktauswurf nach Einschalten
	= "A 1.0" A1.0 -- Y-3 Kontakt-Schieben
	*)
	IO.outY3KontaktSchieben :=	VAT.bAbisoliererLINKSundAUF OR // Abisolierer nach links + Abisolierer auf
								VAT.bCrimpeinheitVOR OR // Crimpeinheit vor
								VAT.bCrimpenZU OR // Crimpen zu
								VAT.bDrahtHalterUndFuehrungAUF OR // Drahthalter + Drahtführung auf
								VAT.bCrZangeAUF_AisolierVOR OR // Crimpzange auf + Abisoliereinheitvor
								VAT.bAusstossenVOR OR // Ausstoßen vor
								VAT.bCrimpeinheitRUECK OR // Crimpeinheit rück
								GVL.tsvKontauswurf.Q ;   // Kontaktauswurf nach Einschalten
								
	(*
	O "M 20.5" M20.5 -- 5---Crimpen zu
	O "M 20.6" M20.6 -- 6---Drahthalter + Drahtführung auf
	UN "M 21.6" M21.6 -- Aktueller Ablauf ohne Crimpen
	O "M 22.6" M22.6 -- Crimpen zu bei Einstellen Leerf-o-Ce
	= "A 1.6" A1.6 -- Y-9 Crimpen zu
	*)
	
	IO.outY9CrimperZU :=	((VAT.bCrimpenZU OR  // Crimpen zu
							VAT.bDrahtHalterUndFuehrungAUF) AND // Drahthalter + Drahtführung auf
								NOT VAT.bAktAblaufOhneCr) OR // Aktueller Ablauf ohne Crimpen
							VAT.bCrimpenZuBeiEinstellen; //Crimpen zu bei Einstellen Leerf-o-Ce	
	(*
	O "M 21.0" M21.0 -- 8---Ausstoßen vor
	O "M 21.1" M21.1 -- 9---Crimpeinheit rück
	O "T 19" T19 -- Kontaktauswurf nach Einschalten
	= "A 0.6" A0.6 -- Y-1 Ausstoßen
	*)
	
	IO.outY1Ausstossen :=	VAT.bAusstossenVOR OR // Ausstoßen vor
							VAT.bCrimpeinheitRUECK OR // Crimpeinheit rück
							GVL.tsvKontauswurf.Q; // Kontaktauswurf nach Einschalten

END_FUNCTION

// ---- POUs/MainPous/FC24_Sortierer/P_Sortierer.TcPOU
PROGRAM P_Sortierer
VAR
END_VAR

(* 
Baustein: FC24 Sortierer
Zeitstempel Code: 25.06.2018 11:16:45
Interface: 27.09.2011 10:59:21
*)

F_Sortierer(); //OK

F_Vereinzelung(); //SV noch den block verwenden

F_Leerfahren(); //OK

END_PROGRAM

// ---- POUs/MainPous/FC24_Sortierer/F_Sortierer.TcPOU
FUNCTION F_Sortierer : BOOL
VAR_INPUT
END_VAR
VAR
	
END_VAR

(* Netzwerk: 1 Sortierer *)


(*
	U "E2_5" E2.5 -- N Magazin gefüllt
	L S5T#100MS
	SA "T 32" T32 -- Verl. E2.5 Magazin gefüllt
*)
GVL.tofMagazGefuellt(IN := GVL.insecMagazinGEFUELLT, PT := T#100MS);
(*	
	U "T 32" T32 -- Verl. E2.5 Magazin gefüllt
	L S5T#1S
	SE "T 33" T33 -- Verl. T32 E2.5 Magazin gefüllt
*)	
GVL.tofMagazGefuellt2(IN := GVL.tofMagazGefuellt.Q, PT := T#1S);	
	
(*	
	L 0 //Sortierer aus
	UN "T 33" T33 -- Verl. T32 E2.5 Magazin gefüllt
	UN "M1.3_Stop" M1.3 -- RS Stop StST
	UN "M8.3CrimpEinr" M8.3 -- Crimpen Einrichten
	UN "M8.4NurAbisolieren" M8.4 -- Nur Abisolieren
	U "T 72" T72 -- Verz. Alles OK von PNOZ PNOZ
	SPBN fh
*)
GVL.TopfWert := 0;

IF	NOT GVL.tofMagazGefuellt2.Q AND //T33
	NOT VAT.bRsStop AND //M1.3 (Unterschied zu "Magazin Leerfahren")
	NOT VAT.bCrimpEinrichten AND //M8.3
	NOT VAT.bNurAbisolieren AND //M8.4
	GVL.tonSAFETYok.Q THEN //T72
	
	(*	
		L "DB6".w132_Sortierer DB6.DBW132 -- Sortierer-Sollwert (Analog)
		L 130
		*I   -- AKKU1 und AKKU2 multiplizieren,  und speichert das Ergebnis in AKKU1
		+ 3000  -- Addiere AKKU1-L und 3000, speichere das Ergebnis in AKKU1-L. 
	*)	
	
	//y=ax+b Ansatz -- NEU-NBT
	GVL.TopfWert := REAL_TO_UINT(GVL.devSortierer.dFakt_A * INT_TO_REAL(DB6.iSortierer) + GVL.devSortierer.dSmd_B);
	
END_IF

(*
fh: T "AW 4" AW4 -- Sortierer
	L 3500
	>I
	U "M9.0MitBlasen" M9.0 -- mit Sortier-Blasen
	= "A 0.1" A0.1 -- Y-11 Blasluft Sortierer
*)

IO.outSollwertRuettelTopf := GVL.TopfWert; //Checken !!! Checken !!! Checken !!!
IF 3500 > GVL.TopfWert THEN
	IO.outY11SortierLuft := VAT.bSortiererBlasen;
END_IF


IF VAT.bSortiererBlasen THEN
	VAT.sortierTextID := 1000;
ELSE
	VAT.sortierTextID := 1001;
END_IF

END_FUNCTION

// ---- POUs/MainPous/FC24_Sortierer/F_Vereinzelung.TcPOU
FUNCTION F_Vereinzelung : BOOL
VAR_INPUT
END_VAR
VAR
	rtrM24_1 : R_TRIG;
	bTmp : BOOL;
	
	svTrg17:R_TRIG;
	svMerker17 : BOOL; //todo: evtl. nach oben in das PRG bubblen lassen.
END_VAR

(* Netzwerk: 2 Vereinzelung *)

(*
U "M 14.0" M14.0 -- A55 Kontakt nicht gefallen
U "T 3" T3 -- Fehler-Kontr.Maschine (keine Bewegung)
U "M 82.5" M82.5 -- +F E2.5 Magazin gefüllt
S "M 23.3" M23.3 -- S&R 2ter Vereinzelungs-Versuch
*)
bTmp := VAT.bA55KontaktNichtGefallen AND GVL.tonFehlerKontrMaschine.Q AND VAT.bFlankeMagazGefuellt;
IF bTmp THEN
	VAT.bSr2terVereinzVersuch := TRUE;
END_IF

(*
U "M 23.3" M23.3 -- S&R 2ter Vereinzelungs-Versuch
L S5T#300MS
SE "T 21" T21 -- Verz. 2ter Vereinzelungs-Versuch
*)
GVL.ton2terVersuch(IN := VAT.bSr2terVereinzVersuch, PT := T#300MS); // war T21

(*
U "T 21" T21 -- Verz. 2ter Vereinzelungs-Versuch
FP "M 24.1" M24.1 -- Positive Flanke, Zuw.v.T21 2ter Vereinzelungs-Versuch
= "M 24.2" M24.2 -- +F 2ter Vereinzelungs-Versuch
*)
//M24.1 ist offensichtlich der Arbeits-Speicher für den Trigger..., Seite 1-28 AWL_d.pdf
rtrM24_1(Clk := GVL.ton2terVersuch.Q);
VAT.bFlk2terVersuch := rtrM24_1.Q;

(*
U "M 21.7" M21.7 -- Kontakt-Anforderung
UN "M 24.2" M24.2 -- +F 2ter Vereinzelungs-Versuch
L S5T#300MS
SV "T 17" T17 -- Vereinzelungs-Zeit, Zeit als Zeit mit verlängertem Impuls starten
*)

//Zeit als Zeit mit verlängertem Impuls TSV
GVL.tsvVereinzelZeit(IN := VAT.bKontaktAnforderung AND NOT VAT.bFlk2terVersuch, PT := T#300MS);

(*
O "T 17" T17 -- Vereinzelungs-Zeit
O "M 23.0" M23.0 -- Takt für Vereinzelung bei Leerfahren
= "A 0.7" A0.7 -- Y-2 Kontakt-Vereinzelung
*)
IO.outY2KontaktVereinzelung := (GVL.tsvVereinzelZeit.Q OR VAT.bTaktVereinzLeerF);

(*
U "E2_0" E2.0 -- L Kontakt gefallen
L S5T#300MS
SE "T 18" T18 -- Verz.v. E2.0 Kontakt gefallen (SE->TON)
*)

//NBT: Warum und so lange??? War 300ms
GVL.tonKontaktIstGefallen(IN := GVL.insecKontaktIstGefallen, PT := T#300MS);
(*
U "T 18" T18 -- Verz.v. E2.0 Kontakt gefallen
R "M 21.7" M21.7 -- Kontakt-Anforderung
*)
IF GVL.tonKontaktIstGefallen.Q THEN
	VAT.bKontaktAnforderung := FALSE;
END_IF

END_FUNCTION

// ---- POUs/MainPous/FC24_Sortierer/F_Leerfahren.TcPOU
FUNCTION F_Leerfahren : BOOL
VAR_INPUT
END_VAR
VAR
END_VAR

(* Netzwerk: 3 Leerfahren *)

(*
	O "M8.1MagLeerf" M8.1 -- Magazin Leerfahren
	O "M8.2SortLeerf" M8.2 -- Sortierer Leerfahren
	S "M 23.1" M23.1 -- Zylinder sollen IN Leerfahrstellung
*)	
IF VAT.bMagazinLeerfahren OR VAT.bSortiererLeerfahren THEN
	VAT.bZylINLeerFahrt := TRUE; //Zylinder sollen IN Leerfahrstellung
END_IF

(*	
	UN "M8.1MagLeerf" M8.1 -- Magazin Leerfahren
	UN "M8.2SortLeerf" M8.2 -- Sortierer Leerfahren
	U "M 23.1" M23.1 -- Zylinder sollen IN Leerfahrstellung
	R "M 23.1" M23.1 -- Zylinder sollen IN Leerfahrstellung
	S "M 23.2" M23.2 -- Zylinder sollen AUS Leerfahrstellung
*)
IF NOT VAT.bMagazinLeerfahren AND
	NOT VAT.bSortiererLeerfahren AND
	VAT.bZylINLeerFahrt THEN
	
	VAT.bZylINLeerFahrt := FALSE;
	VAT.bZylAUSLeerFahrt := TRUE;
END_IF

(*	
	O "M 23.0" M23.0 -- Takt für Vereinzelung bei Leerfahren
	SPBN kl
*)

IF NOT VAT.bTaktVereinzLeerF THEN
	RETURN;
END_IF

(*	
	U "T 41" T41 -- Takt für Magazin leerfahren
	SPB kl
*)
GVL.tofMagazLeerFahr(IN := FALSE, PT := T#500MS);
IF GVL.tofMagazLeerFahr.Q THEN
	RETURN;
END_IF

(*
	L S5T#500MS
	SA "T 41" T41 -- Takt für Magazin leerfahren
	CLR
	SA "T 41" T41 -- Takt für Magazin leerfahren
	
	UN "M 23.0" M23.0 -- Takt für Vereinzelung bei Leerfahren
	= "M 23.0" M23.0 -- Takt für Vereinzelung bei Leerfahren
*)
GVL.tofMagazLeerFahr(IN := TRUE, PT := T#500MS);
VAT.bTaktVereinzLeerF := NOT VAT.bTaktVereinzLeerF;

(*
kl: BLD 130
*)

END_FUNCTION

// ---- POUs/MainPous/FC3_FehlerAllg/P_FehlerAllgemein.TcPOU
PROGRAM P_FehlerAllgemein
VAR
	fbKontrolleEndschalter : FB_KontrolleEndschalter;
END_VAR

(* Baustein: FC3 Fehlererkennung allgemein *)
(* Name: FEHL_ERK *)
(* Zeitstempel Code: 19.10.2011 10:02:13 *)
(* Interface: 09.07.2010 10:27:01 *)

F_KontrollZeiten();

F_Doppelmeldung(); //OK

F_AusloeseschalterDauermeldung(); //noch ohne Wirkung

fbKontrolleEndschalter(errorOffset := 600); //OK - 600er ID-Bereich

//F_Aufstarten();

F_FehlerAufgetreten();
(*
IF F_FehlerAufgetreten() THEN
	F_StoerungsbitsAuswerten();
END_IF
*)

END_PROGRAM

// ---- POUs/MainPous/FC3_FehlerAllg/FB_KontrolleEndschalter.TcPOU
FUNCTION_BLOCK FB_KontrolleEndschalter 
VAR_INPUT
	errorOffset : WORD := 600;
END_VAR
VAR_OUTPUT
	bError : BOOL;
	nErrNo : WORD;
END_VAR
VAR
END_VAR

(* Netzwerk: 4 Kontr. Endschalter *)
(*
U "T 3" T3 -- Fehler-Kontr.Maschine (keine Bewegung)
U "T 72" T72 -- Verz. Alles OK von PNOZ
SPBN kk
*)
nErrNo := 0;
bError := FALSE;
IF NOT (GVL.tonFehlerKontrMaschine.Q AND GVL.tonSAFETYok.Q) THEN
	RETURN;
END_IF

(*
UN "A 1.7" A1.7 -- Y-10 Drahthalter+Führung zu
UN "E1_0" E1.0 -- R Drahthalter offen
S "F40 E1.0f" M104.0 -- Drahthalter nicht offen
*)
IF NOT IO.outY10DrahthaltFuehrungZU AND NOT GVL.insecDrahthalterIstOffen THEN
	GVL.errs.DrahthltNichtOffen := TRUE;
	nErrNo := errorOffset;
END_IF
(*
U "A 1.7" A1.7 -- Y-10 Drahthalter+Führung zu
U "E1_0" E1.0 -- R Drahthalter offen
S "F41 E1.0nw" M104.1 -- Drahthalter nicht zu
*)
IF IO.outY10DrahthaltFuehrungZU AND GVL.insecDrahthalterIstOffen THEN
	GVL.errs.DrahthltNichtZu := TRUE;
	nErrNo := errorOffset + 1;
END_IF


(*
UN "A 1.3" A1.3 -- Y-6 Abisolierer zu
U "E1_2" E1.2 -- N Abisolierer zu
S "F43 E1.2nw" M104.3 -- Abisolierer nicht offen
*)
IF NOT IO.outY6AbisoliererZU AND GVL.insecAbisoliererIstZU THEN
	GVL.errs.AbisolierNichtOffen := TRUE;
	nErrNo := errorOffset + 3;
END_IF


(*
U "A 1.3" A1.3 -- Y-6 Abisolierer zu
UN "E1_2" E1.2 -- N Abisolierer zu
S "F44 E1.2f" M104.4 -- Abisolierer nicht zu
*)
IF  IO.outY6AbisoliererZU AND NOT GVL.insecAbisoliererIstZU THEN
	GVL.errs.AbisolierNichtZu := TRUE;
	nErrNo := errorOffset + 4;
END_IF

(*
UN "A 1.5" A1.5 -- Y-8 Abisolierer rück
UN "E1_3" E1.3 -- R Abisolierer vorn
S "F46 E1.3f" M104.6 -- Abisolierer nicht vorn
*)
IF NOT IO.outY8AbisoliererRUECK AND NOT GVL.insecAbisoliererIstVORN THEN
	GVL.errs.AbisolierNichtVorn := TRUE;
	nErrNo := errorOffset + 6;
END_IF


(*
U "A 1.5" A1.5 -- Y-8 Abisolierer rück
UN "E1_4" E1.4 -- R Abisolierer rück (abisoliert)
S "F47 E1.4f" M104.7 -- Abisolierer nicht rück (abisoliert)
*)
IF IO.outY8AbisoliererRUECK AND NOT GVL.insecAbisoliererIstRUECK THEN
	GVL.errs.AbisolierNichtRueck := TRUE;
	nErrNo := errorOffset + 7;
END_IF


(*
U "A 1.2" A1.2 -- Y-5 Abisolierer nach links+Abdeckung zu
UN "E1_5" E1.5 -- R Abisolierer links (aus Arbeitsraum)
S "F50 E1.5f" M105.0 -- Abisolierer nicht links (aus Arbeitsraum)
*)
IF IO.outY5AbisolierNachLINKS AND NOT GVL.insecAbisoliererIstLINKS THEN
	GVL.errs.AbisolierNichtLinks := TRUE;
	nErrNo := errorOffset + 8;	
END_IF


(*
UN "A 1.2" A1.2 -- Y-5 Abisolierer nach links+Abdeckung zu
U "E1_5" E1.5 -- R Abisolierer links (aus Arbeitsraum)
S "F51 E1.5nw" M105.1 -- Abisolierer nicht rechts
*)
IF NOT IO.outY5AbisolierNachLINKS AND GVL.insecAbisoliererIstLINKS THEN
	GVL.errs.AbisolierNichtRechts := TRUE;
	nErrNo := errorOffset + 9;
END_IF


(*
U "A 1.6" A1.6 -- Y-9 Crimpen zu
UN "E1_6" E1.6 -- N Crimpzange zu
S "F53 E1.6f" M105.3 -- Crimpzange nicht zu
*)
IF IO.outY9CrimperZU AND NOT GVL.insecCrimpZangeIstZU THEN
	GVL.errs.CrimpZangeNichtZu := TRUE;
	nErrNo := errorOffset + 11;
END_IF


(*
UN "A 1.6" A1.6 -- Y-9 Crimpen zu
UN "E1_7" E1.7 -- R Crimpzange offen
S "F54 E1.7f" M105.4 -- Crimpzange nicht offen
*)
IF NOT IO.outY9CrimperZU AND NOT GVL.insecCrimpZangeIstOFFEN THEN
	GVL.errs.CrimpZangeNichtOffen := TRUE;
	nErrNo := errorOffset + 12;
END_IF


(* ToDo:
errKontaktNichtGefallen : BOOL; //(ehem. M105.5) !! nur xls File !! --
*)

//NEU
GVL.tonKontaktIstZuLangeEin(IN := GVL.insecKontaktIstGefallen, PT := T#2S);
IF GVL.tonKontaktIstZuLangeEin.Q THEN
	GVL.errs.DauerMlgKontaktGefallen := TRUE; //(ehem. 105.6) !! nur xls File !! --
	nErrNo := errorOffset + 14;
END_IF
(*
U "A 1.1" A1.1 -- Y-4 Crimpeinheit vor
UN "E2_1" E2.1 -- R Crimpeinheit vorn
S "F60 E2.1f" M106.0 -- Crimpeinheit nicht vorn
*)
IF IO.outY4CrimpEinheitVOR AND NOT GVL.insecCrimpEinheitIstVORN THEN
	GVL.errs.CrimpeinheitNichtVorn := TRUE;
nErrNo := errorOffset + 16;	
END_IF


(*
UN "A 1.1" A1.1 -- Y-4 Crimpeinheit vor
UN "E2_4" E2.4 -- R Crimpeinheit rück
S "F61 E2.4f" M106.1 -- Crimpeinheit nicht rück
*)
IF NOT IO.outY4CrimpEinheitVOR AND NOT GVL.insecCrimpEinheitIstRUECK THEN
	GVL.errs.CrimpeinheitNichtRueck := TRUE;
nErrNo := errorOffset + 17;	
END_IF


(*
U "A 1.0" A1.0 -- Y-3 Kontakt-Schieben
UN "E2_2" E2.2 -- R Kontakt-Schieben vorn
S "F62 E2.2f" M106.2 -- Kontakt-Schieben nicht vorn
*)
IF IO.outY3KontaktSchieben AND NOT GVL.insecKontaktSchiebenVORN THEN
	GVL.errs.KontaktSchiebenNichtVorn := TRUE;
	nErrNo := errorOffset + 18;
END_IF


(*
UN "A 1.0" A1.0 -- Y-3 Kontakt-Schieben
U "E2_2" E2.2 -- R Kontakt-Schieben vorn
S "F63 E2.2nw" M106.3 -- Kontakt-Schieben nicht rück
*)
IF NOT IO.outY3KontaktSchieben AND GVL.insecKontaktSchiebenVORN THEN
	GVL.errs.KontaktSchiebenNichtRueck := TRUE;
	nErrNo := errorOffset + 19;
END_IF


(*
U "A 0.6" A0.6 -- Y-1 Ausstoßen
UN "E2_3" E2.3 -- R Ausstoßen vorn
S "F64 E2.3f" M106.4 -- Ausstoßen nicht vorn
*)
IF IO.outY1Ausstossen AND NOT GVL.insecAusstossenVORN THEN
	GVL.errs.AusstossenNichtVorn := TRUE;
	nErrNo := errorOffset + 20;	
END_IF


(*
UN "A 0.6" A0.6 -- Y-1 Ausstoßen
U "E2_3" E2.3 -- R Ausstoßen vorn
S "F65 E2.3nw" M106.5 -- Ausstoßen nicht rück
*)
IF NOT IO.outY1Ausstossen AND GVL.insecAusstossenVORN THEN
	GVL.errs.AusstossenNichtRueck := TRUE;
	nErrNo := errorOffset + 21;
END_IF


//NBT-NEU
IF nErrNo <> 0 THEN
	bError := TRUE;
END_IF

(*
kk: BLD 130
*)

END_FUNCTION_BLOCK

// ---- POUs/MainPous/FC3_FehlerAllg/F_KontrollZeiten.TcPOU
FUNCTION F_KontrollZeiten : BOOL
VAR_INPUT
END_VAR
VAR
	bTmp : BOOL;
	localWord:WORD;
END_VAR

(* Netzwerk: 1 *** Kontroll-Zeiten *)

//ToDo: den Sinn der Aktion herausbekommen...
//evtl. Bitmuster auf dem AW erkennen...
(*
L AW 0 -- Akku 1 nach Akku 2, dann AW0 in Akku 1 -- AW0 offensichtlich Ausgangswort 0
T LW 0 -- Akku 1 nach LW 0 -- Ausgangswort0 in LW 0 speichern
L "DB6".d408 DB6.DBD408 -- Zuw.v. AW0 -- Akku 1 nach Akku 2, dann "DB6".d408 in Akku 1

L LD 0 -- Akku 1 nach Akku 2, dann LD 0 in Akku 1 -- Frage, was steht in LD 0 (Lokaldaten-Doppelwort (LD))

T "DB6".d408 DB6.DBD408 -- Zuw.v. AW0 -- T beeinflusst nichts...

-- [XOD] ... Bei der Verknüpfung von Doppelwörtern wird der Inhalt von AKKU 2 mit dem Inhalt von AKKU 1 verknüpft.
--  Das Verknüpfungsergebnis wird in AKKU 1 gespeichert, wobei der alte Inhalt überschrieben wird.

XOD

L 2# 11000000 11111111 00000000 00000000 -- Akku 1 nach Akku 2, dann Zahl in Akku 1
UD -- UND-Doppelwort
L 0
==D
*)

//Versuch...die Maske L 2# 110... kann wahrscheinlich entfallen, da ich das beim Füllen von IO.outWord0 schon
//berücksichtige NBT 2021-01-28

bTmp := (DB6.outWordAlt XOR IO.outWord0) <> 0; //ToDo: ergebnis dieser Aktion

(*
L S5T#1S200MS
SE "T 3" T3 -- Fehler-Kontr.Maschine (keine Bewegung) -- Zeit mit Einschaltverzögerung starten
L S5T#1S600MS
SE "T 15" T15 -- Verz. Endschalter-Brückung StSt *)

GVL.tonFehlerKontrMaschine( IN := bTmp, PT := T#1S200MS);

GVL.tonEndschalterBrueck( IN := bTmp, PT := T#1S600MS);

DB6.outWordAlt := IO.outWord0;

END_FUNCTION

// ---- POUs/MainPous/FC3_FehlerAllg/F_Doppelmeldung.TcPOU
FUNCTION F_Doppelmeldung : BOOL
VAR_INPUT
END_VAR
VAR
END_VAR

(* Netzwerk: 2 Doppelmeldung *)

(*
U "E1_3" E1.3 -- R Abisolierer vorn
U "E1_4" E1.4 -- R Abisolierer rück (abisoliert)
S "F45 E1.3+E1.4" M104.5 -- Doppelmeldung Abisolierer vorn+rück *)
IF GVL.insecAbisoliererIstVORN AND GVL.insecAbisoliererIstRUECK THEN
	GVL.errs.DoppelMlgAbisoVornRueck := TRUE;
END_IF


(*
U "E1_6" E1.6 -- N Crimpzange zu
U "E1_7" E1.7 -- R Crimpzange offen
S "F52 E1.6+E1.7" M105.2 -- Doppelmeldung Crimpzange zu+offen
*)
IF GVL.insecCrimpZangeIstZU AND GVL.insecCrimpZangeIstOFFEN THEN
	GVL.errs.DoppelMlgCrimpzZuOffen := TRUE;
END_IF


(*
U "E2_1" E2.1 -- R Crimpeinheit vorn
U "E2_4" E2.4 -- R Crimpeinheit rück
S "F57 E2.1+E2.4" M105.7 -- Doppelmeldung Crimpeinheit vorn+rück
*)
IF GVL.insecCrimpEinheitIstVORN AND GVL.insecCrimpEinheitIstRUECK THEN
	GVL.errs.DoppelMlgCrimpEinhVornZurueck := TRUE;
END_IF

END_FUNCTION

// ---- POUs/MainPous/FC3_FehlerAllg/F_AusloeseschalterDauermeldung.TcPOU
FUNCTION F_AusloeseschalterDauermeldung : BOOL
VAR_INPUT
END_VAR
VAR
	tmp:BOOL;
END_VAR

(* Netzwerk: 3 Auslöseschalter Dauermeldung *)

(*
U "M 22.7" M22.7 -- Endstellung
U "E1_1" E1.1 -- N Auslöseschalter
L S5T#2S
SE "T 16" T16 -- Kontr.Auslöseschalter Dauermeldung
U "T 16" T16 -- Kontr.Auslöseschalter Dauermeldung
S "F42 E1.1nw" M104.2 -- Auslöseschalter Dauermelung
*)
//SE == TON

GVL.tonAusloesDauermld(IN := VAT.bEndstellung AND IO.inAusloeseSchalter, PT := T#2S);
IF GVL.tonAusloesDauermld.Q THEN
	GVL.errs.AusloesSchaltDauerMldg := TRUE;
END_IF

END_FUNCTION

// ---- POUs/MainPous/FC3_FehlerAllg/F_FehlerAufgetreten.TcPOU
FUNCTION F_FehlerAufgetreten : BOOL
(* Soll eine Fehlerauswertung gemacht werden oer nicht *)
VAR_INPUT
END_VAR
VAR
	akku : DWORD;
END_VAR

(* Netzwerk: 6 *** Fehler aufgetreten ? *)

(*
L MD 100
L MD 104
OD -- ODER-Doppelwort
L MD 108
OD -- ODER-Doppelwort
L 0
<>D -- 	AKKU2 ungleich AKKU1 [DWORD], also wenn die Merker Fehler enthalten...ist VKE 1
= "M0.7" M0.7 -- Störung aufgetreten (gesammelt)
*)
GVL.errsAsDword := F_GetErrorsAsDWORD(errStruct := GVL.errs);
//...größerer Umbau gegenüber altem AWL-Programm, aber vom Prinzip her gleich.
VAT.bSammelStoerung := GVL.errsAsDword <> 0; //Sammel-Störung

(*
SPB X027 -- Springe wenn VKE = 1, ... zu X027, also überspringe RETURN.
BEA -- Bausteinende absolut, im Falle KEINES Fehlers: Keine Fehlerbitauswertung
*)
IF NOT VAT.bSammelStoerung THEN
	F_FehlerAufgetreten := FALSE;
	RETURN;
END_IF

//...jetzt noch nachsehen, ob SAFETY ok ist...
(*
X027: UN "T 72" T72 -- Verz. Alles OK von SAFETY (früher PNOZ), Fage ist SAFETY FALSE ?
BEB -- Bausteinende bedingt, Wenn SAFETY auch FALSE: auch Keine Fehlerbitauswertung 
*)

IF NOT GVL.tonSAFETYok.Q THEN
	F_FehlerAufgetreten := FALSE; //Wenn SAFETY = FALSE, Keine Fehlerbitauswertung 
	RETURN;
END_IF

F_FehlerAufgetreten := TRUE; //Auswertung fahren...

END_FUNCTION

// ---- POUs/MainPous/FC3_FehlerAllg/F_GetErrorsAsDWORD.TcPOU
FUNCTION F_GetErrorsAsDWORD : DWORD
VAR_INPUT
	errStruct : DUT_Errors; 
END_VAR
VAR
	pTmp : POINTER TO DWORD;
END_VAR


pTmp := ADR(errStruct);


//pTmp := ADR(errStruct.DrahthltNichtOffen); //erstes Element von err : DUT_Errors

F_GetErrorsAsDWORD := pTmp^;

END_FUNCTION

// ---- POUs/MainPous/FC95_StatusAnzeige/P_StatusAnzeige.TcPOU
PROGRAM P_StatusAnzeige
VAR
END_VAR

(*
Baustein: FC95 Status-Anzeige
Zeitstempel Code: 09.12.2014 10:56:48
Interface: 09.07.2010 10:27:01
*)

//NBT-NEU

GVL.zeigeFehler := (P_Ablauf.fbAllesInSollpos.bError AND NOT P_Ablauf.fbAllesInSollpos.bErrMute)
					OR P_FehlerAllgemein.fbKontrolleEndschalter.bError;


(* Netzwerk: 1 *)

//ToDo: Noch keine Ahnung, was das tun soll...
(*
L "DB6".d42 DB6.DBB42	-- Eingangs-Byte-Select Status

// https://www.sps-forum.de/simatic/81525-variabler-array-index-awl.html
//Beispiel:
//L #index    // 1..8 (aus MB23)
//+ -1        // --> 0..7
//SLD 3       // * 8 --> Byteadresse.0 -- Array_Index: 0 ... (muß * 8, weil Bit-Adressen adressiert werden, wir aber die Byte-Adresse brauchen)
			  //  Element_Größe: 1 = Byte / 2 = Word / 4 = DWord
			  

SLW 3 					-- Schiebt Wort um 3 bit nach links, bzw. multipliziert den Wert im Akku mit 8. Siehe oben...
// * 1 für Byte-Array rechnen nicht nötig

LAR1 					-- Akku als Zeiger in Adressregister 1 laden
L EB [AR1,P#0.0] 		-- Lade Eingangsbyte, Adressregister 1 mit Offset 0.0 adressiert
T "DB6".d40 DB6.DBB40 	-- 8*Eingangs-Bit Status
*)

(*
L "DB6".d46 DB6.DBB46 -- Ausgangs-Byte-Select Status
SLW 3
LAR1
L "DB6".d43 DB6.DBB43 -- Zuw.v.DBB46 Status
L "DB6".d46 DB6.DBB46 -- Ausgangs-Byte-Select Status
T "DB6".d43 DB6.DBB43 -- Zuw.v.DBB46 Status
==I
= L 0.0  -- L 0.0 ist das erste bit aus den lokaldaten
*)



(*
L "DB6".d45 DB6.DBB45 -- Zuw.vom selectierten Ausgangs-Byte Status
L AB [AR1,P#0.0]	  -- Lade Ausgangsbyte
T "DB6".d45 DB6.DBB45 -- Zuw.vom selectierten Ausgangs-Byte Status
<>I
R L 0.0
*)



(*
//https://www.sps-forum.de/simatic/6451-awl-anweisung-verstehen.html
//L 0.0 ist das erste bit aus den lokaldaten.
//Auf jeden Fall ist das keine saubere Arbeit. Siemens macht sowas gerne beim umschalten von KOP/FUP in AWL,
//aber ein Programmierer sollte das nicht tun.

U L 0.0
SPBN s1
*)

(*
	L "DB6".d44 DB6.DBB44 -- 8*Ausgangs-Bit Status
	T AB [AR1,P#0.0]
*)
	
(*	
s1: L AB [AR1,P#0.0]
	T "DB6".d44 DB6.DBB44 -- 8*Ausgangs-Bit Status
	L "DB6".d50 DB6.DBB50 -- Merker-Byte-Select Status
	SLW 3
	LAR1
	L "DB6".d47 DB6.DBB47 -- Zuw.v.DBB50 Status
	L "DB6".d50 DB6.DBB50 -- Merker-Byte-Select Status
	T "DB6".d47 DB6.DBB47 -- Zuw.v.DBB50 Status
	==I
	= L 0.0
	L "DB6".d49 DB6.DBB49 -- Zuw.vom selectierten Merker-Byte Status
	L MB [AR1,P#0.0]
	T "DB6".d49 DB6.DBB49 -- Zuw.vom selectierten Merker-Byte Status
	<>I
	R L 0.0
	U L 0.0
	SPBN s2
	L "DB6".d48 DB6.DBB48 -- 8*Merker-Bit Status
	T MB [AR1,P#0.0]
s2: L MB [AR1,P#0.0]
	T "DB6".d48 DB6.DBB48 -- 8*Merker-Bit Status
	L MW [AR1,P#0.0]
	T "DB6".d52 DB6.DBW52 -- Wert vom selectierten Merker-Byte Status
*)

;

END_PROGRAM

// ---- POUs/MainPous/FC2_Betriebsarten/P_OutputHandling.TcPOU
PROGRAM P_OutputHandling
VAR
	outWordOld : WORD;
END_VAR


	IO.outY1Ausstossen := IO.outY1Ausstossen OR DB6.frceY1Ausstossen;
	IO.outY2KontaktVereinzelung := IO.outY2KontaktVereinzelung OR DB6.frceY2KontaktVereinzelung; //EL1809-A1.7
	IO.outY3KontaktSchieben := IO.outY3KontaktSchieben OR DB6.frceY3KontaktSchieben; //EL1809-A1.8
	IO.outY4CrimpEinheitVOR := IO.outY4CrimpEinheitVOR OR DB6.frceY4CrimpEinheitVOR;//EL1809-A1.9
	IO.outY5AbisolierNachLINKS := IO.outY5AbisolierNachLINKS OR DB6.frceY5AbisolierNachLINKS;//EL1809-A1.10
	IO.outY6AbisoliererZU := IO.outY6AbisoliererZU OR DB6.frceY6AbisoliererZU; //EL1809-A1.11
	IO.outY7AbfallRUNTER := IO.outY7AbfallRUNTER OR DB6.frceY7AbfallRUNTER; //EL1809-A1.12
	IO.outY8AbisoliererRUECK := IO.outY8AbisoliererRUECK OR DB6.frceY8AbisoliererRUECK; //EL1809-A1.13
	IO.outY9CrimperZU := IO.outY9CrimperZU OR DB6.frceY9CrimperZU; //EL1809-A1.14
	IO.outY10DrahthaltFuehrungZU := IO.outY10DrahthaltFuehrungZU OR DB6.frceY10DrahthaltFuehrungZU; //EL1809-A1.15
	IO.outY11SortierLuft := IO.outY11SortierLuft OR DB6.frceY11SortierLuft; //EL1809-A1.5
	
	IO.outWord0 :=
		
	SHL(BOOL_TO_WORD(IO.outY11SortierLuft		), 5) + //EL1809-A1.5
	SHL(BOOL_TO_WORD(IO.outY1Ausstossen			), 6) + //EL1809-A1.6
	SHL(BOOL_TO_WORD(IO.outY2KontaktVereinzelung), 7) + //EL1809-A1.7
	SHL(BOOL_TO_WORD(IO.outY3KontaktSchieben	), 8) + //EL1809-A1.8
	SHL(BOOL_TO_WORD(IO.outY4CrimpEinheitVOR	), 9) + //EL1809-A1.9
	SHL(BOOL_TO_WORD(IO.outY5AbisolierNachLINKS	), 10) + //EL1809-A1.10
	SHL(BOOL_TO_WORD(IO.outY6AbisoliererZU		), 11) + //EL1809-A1.11
	SHL(BOOL_TO_WORD(IO.outY7AbfallRUNTER		), 12) + //EL1809-A1.12
	SHL(BOOL_TO_WORD(IO.outY8AbisoliererRUECK	), 13) + //EL1809-A1.13
	SHL(BOOL_TO_WORD(IO.outY9CrimperZU			), 14) + //EL1809-A1.14
	SHL(BOOL_TO_WORD(IO.outY10DrahthaltFuehrungZU),15); //EL1809-A1.15
	
	
	IF outWordOld <> IO.outWord0 THEN
		MAIN.M_Log(reqLevel:=CVL.TRACE, objectName:= 'OUT', sMsg:= '--------',errNo := 16#FFFFFFFF);
		//MAIN.M_Log(reqLevel:=CVL.TRACE, objectName:= 'OUT', sMsg:= 'Y11SortierLuft', errNo:= BOOL_TO_UDINT(IO.outY11SortierLuft));
		MAIN.M_Log(reqLevel:=CVL.TRACE, objectName:= 'OUT', sMsg:= 'Y1Ausstossen', errNo:= BOOL_TO_UDINT(IO.outY1Ausstossen));
		MAIN.M_Log(reqLevel:=CVL.TRACE, objectName:= 'OUT', sMsg:= 'Y2KontaktVereinzelung', errNo:= BOOL_TO_UDINT(IO.outY2KontaktVereinzelung));
		MAIN.M_Log(reqLevel:=CVL.TRACE, objectName:= 'OUT', sMsg:= 'Y3KontaktSchieben', errNo:= BOOL_TO_UDINT(IO.outY3KontaktSchieben));
		MAIN.M_Log(reqLevel:=CVL.TRACE, objectName:= 'OUT', sMsg:= 'Y4CrimpEinheitVOR', errNo:= BOOL_TO_UDINT(IO.outY4CrimpEinheitVOR));
		MAIN.M_Log(reqLevel:=CVL.TRACE, objectName:= 'OUT', sMsg:= 'Y5AbisolierNachLINKS', errNo:= BOOL_TO_UDINT(IO.outY5AbisolierNachLINKS));
		MAIN.M_Log(reqLevel:=CVL.TRACE, objectName:= 'OUT', sMsg:= 'Y6AbisoliererZU', errNo:= BOOL_TO_UDINT(IO.outY6AbisoliererZU));
		MAIN.M_Log(reqLevel:=CVL.TRACE, objectName:= 'OUT', sMsg:= 'Y7AbfallRUNTER', errNo:= BOOL_TO_UDINT(IO.outY7AbfallRUNTER));
		MAIN.M_Log(reqLevel:=CVL.TRACE, objectName:= 'OUT', sMsg:= 'Y8AbisoliererRUECK', errNo:= BOOL_TO_UDINT(IO.outY8AbisoliererRUECK));
		MAIN.M_Log(reqLevel:=CVL.TRACE, objectName:= 'OUT', sMsg:= 'Y9CrimperZU', errNo:= BOOL_TO_UDINT(IO.outY9CrimperZU));
		MAIN.M_Log(reqLevel:=CVL.TRACE, objectName:= 'OUT', sMsg:= 'Y10DrahthaltFuehrungZU', errNo:= BOOL_TO_UDINT(IO.outY10DrahthaltFuehrungZU));
	
	END_IF

outWordOld := IO.outWord0;

END_PROGRAM

// ---- POUs/HMI/P_HmiHandling.TcPOU
PROGRAM P_HmiHandling
VAR
	ntClosePlcHmi : NT_StartProcess;
	bClose : BOOL := FALSE;
END_VAR


ntClosePlcHmi(
	NETID:='' , 
	PATHSTR:='C:\Windows\System32\cmd.exe' , 
	DIRNAME:='C:\Windows\System32' , 
	COMNDLINE:='/c "C:\HMI\ClosePlcHmi.cmd"' , 
	START:=bClose , 
	TMOUT:=T#5S ,
 
	BUSY=> , 
	ERR=> , 
	ERRID=> );

END_PROGRAM

// ---- POUs/MainPous/FC3_FehlerAllg/F_Aufstarten.TcPOU
FUNCTION F_Aufstarten : BOOL
VAR_INPUT
END_VAR
VAR
END_VAR

(* Netzwerk: 5 Aufstarten *)

(*
Die Operation SPA verlangt einen absoluten unbedingten Sprung ohne irgendwelche Bedingungen. SPA ist nicht abhängig vom Signalwert eines Bits
im Statuswort oder vom VKE der vorhergehenden Verknüpfung. Das Anwenderprogramm wird an der angegebenen Sprungmarke weiter abgearbeitet.
Gesprungen werden kann vorwärts und rückwärts, das Sprungziel muss allerdings im gleichen Baustein liegen wie der Aufruf der Sprungoperation
SPA und darf nur einmal vorhanden sein.
*)
//SPA mie -- Springe absolut
RETURN;

GVL.tonTasteStart(IN := IO.inStart, PT := T#2S);

IF GVL.tonTasteStart.Q THEN
	F_ResetErrors();
	(* GVL.MD100 := 0;
	GVL.MD104 := 0;
	GVL.MD108 := 0; 
	GVL.MD112 := 0;
	GVL.MD116 := 0; 
	GVL.MD120 := 0; *)
END_IF
(*
U "E0_0" E0.0 -- Taste Start
L S5T#2S
SE T 11
U T 11
SPB mie -- Springe wenn VKE = 1
L 0
T MD 100
T MD 104
T MD 108
T MD 112
T MD 116
T MD 120
mie: BLD 130
*)

END_FUNCTION

// ---- POUs/Helper/FB_CalcXY.TcPOU
FUNCTION_BLOCK FB_CalcXY
(* Berechnung des a und b Wertes für die Linearisierung Y=ax+b *)
VAR_INPUT
     Dev : POINTER TO DUT_Device;
END_VAR
VAR_OUTPUT

END_VAR 
VAR

END_VAR

(* prevent Div By Zero *)

Dev^.dFakt_A := 1;
Dev^.dSmd_B := 0;

IF (Dev^.rIN_HI - Dev^.rIN_LO) = 0 THEN
     RETURN;
END_IF

Dev^.dFakt_A :=  UINT_TO_REAL(Dev^.nOUT_HI - Dev^.nOUT_LO ) / (Dev^.rIN_HI - Dev^.rIN_LO);
Dev^.dSmd_B := Dev^.nOUT_LO - (Dev^.rIN_LO * Dev^.dFakt_A);

END_FUNCTION_BLOCK

// ---- POUs/Language/P_SaveCurrentLanguage.TcPOU
PROGRAM P_SaveCurrentLanguage
VAR
END_VAR

RVL.currLanguage := VisuElems.CurrentLanguage;

MAIN.M_Log(reqLevel:=CVL.INFO, objectName:= 'P_SaveCurrentLanguage', sMsg:=RVL.currLanguage, errNo:= 0);

END_PROGRAM

// ---- POUs/MainPous/F20_Ablauf/AusstossVerzoegerung/P_DecAusStossV.TcPOU
PROGRAM P_DecAusStossV
VAR
END_VAR

IF DB6.rAusstossverz >= 0.1 THEN
	DB6.rAusstossverz := DB6.rAusstossverz - 0.1;
	DB6.nAusstossverz := REAL_TO_INT(DB6.rAusstossverz * 1000);
END_IF

END_PROGRAM

// ---- POUs/MainPous/F20_Ablauf/AusstossVerzoegerung/P_IncAusstossV.TcPOU
PROGRAM P_IncAusstossV
VAR
END_VAR

IF DB6.rAusstossverz < 0.91 THEN
	DB6.rAusstossverz := DB6.rAusstossverz + 0.1;
	DB6.nAusstossverz := REAL_TO_INT(DB6.rAusstossverz * 1000);
END_IF

END_PROGRAM

// ---- POUs/MainPous/F20_Ablauf/DrahtHalterDruck/P_DecDruck.TcPOU
PROGRAM P_DecDruck
VAR
END_VAR

IF DB6.rDrahthalterSchliessdruck > 0.9 THEN
	DB6.rDrahthalterSchliessdruck := DB6.rDrahthalterSchliessdruck - 0.5;
END_IF

END_PROGRAM

// ---- POUs/MainPous/F20_Ablauf/DrahtHalterDruck/P_IncDruck.TcPOU
PROGRAM P_IncDruck
VAR
END_VAR

IF DB6.rDrahthalterSchliessdruck < 5.9 THEN
	DB6.rDrahthalterSchliessdruck := DB6.rDrahthalterSchliessdruck + 0.5;
END_IF

END_PROGRAM

// ---- POUs/MainPous/F20_Ablauf/SollwertRuettelTopf/P_DecSollRuettel.TcPOU
PROGRAM P_DecSollRuettel
VAR
END_VAR

IF DB6.iSortierer > 0 THEN
	DB6.iSortierer := DB6.iSortierer - 1;
END_IF

END_PROGRAM

// ---- POUs/MainPous/F20_Ablauf/SollwertRuettelTopf/P_IncSollRuettel.TcPOU
PROGRAM P_IncSollRuettel
VAR
END_VAR

IF DB6.iSortierer < 100 THEN
	DB6.iSortierer := DB6.iSortierer + 1;
END_IF

END_PROGRAM

// ---- POUs/MainPous/FC3_FehlerAllg/F_StoerungsbitsAuswerten.TcPOU
FUNCTION F_StoerungsbitsAuswerten : BOOL
VAR_INPUT
END_VAR
VAR
	x:BOOL;
	akku1 : WORD;
	wLocal2 : WORD;
	wLocal4 : WORD;
END_VAR

(* Netzwerk: 7 Störungsbits auswerten und Reset (für Ziffern-Display) *)

(* 
	L 110 //** höchste auszuwertende Wort-Adresse
*)
akku1 := 110;
(*	
Sar1: T LW 2 //Abwärts-Zähler Wort-Adresse
	SLW 3  -- Schiebe Wort nach links
	LAR1
	L MW [AR1,P#0.0]
	T LW 4 //enthält Bits vom aktuellen Störungs-Wort
	L 0
	<>I
	SPB Sar2+
	L 100 //** niedrigste auszuwertende Wort-Adresse
	L LW 2 //Abwärts-Zähler Wort-Adresse
	>=I
	SPB Sar6
	DEC 2
	SPA Sar1 -- Springe absolut
*)

(*
x := TRUE;	
WHILE x = TRUE DO
	wLocal2 := akku1;	
	akku1 := akku1 * 8;



END_WHILE
*)


	
(*	
Sar2: L 2#11111110111111111111111011111111
	T LD 6 //Schiebe-Maske
	L 18
	T LW 0 //Abwärts-Zähler Bit-Adresse
Sar3: L LW 0 //Abwärts-Zähler Bit-Adresse
	DEC 1
	T LW 0 //Abwärts-Zähler Bit-Adresse
	L 9
	<>I
	SPB Sar4
	L 7
	T LW 0 //Abwärts-Zähler Bit-Adresse
Sar4: L LD 6 //Schiebe-Maske
	SRD 1
	T LD 6 //Schiebe-Maske
	L LW 4 //enthält Bits vom aktuellen Störungs-Wort
	L LW 8 //16 Bit rechts der Schiebe-Maske
	UW
	==I
SPB Sar3
	UN "M 6.0" M6.0 -- +F Reset-Button
	SPB Sar5
	L LW 2 //Abwärts-Zähler Wort-Adresse
	SLW 3
	LAR1
	TAK
	T MW [AR1,P#0.0]
Sar5: L LW 2 //Abwärts-Zähler Wort-Adresse
	DEC 100
	L 10
	*I
	L LW 0 //Abwärts-Zähler Bit-Adresse
	+I
	T "DB6".w226_Betr_Anz_Wert DB6.DBW226 -- Betriebs-Anzeige-Wert
Sar6: BLD 130
*)
;

END_FUNCTION

// ---- POUs/MainPous/FC4_TpKommunikation/F_AnzeigeSollpositionsFehler.TcPOU
FUNCTION_BLOCK F_AnzeigeSollpositionsFehler 
VAR_INPUT
	enable : BOOL;
	errNo : WORD;
	idOffset : WORD; 
END_VAR
VAR_OUTPUT
	errID : WORD;
END_VAR
VAR
	//wait : TON;
END_VAR

errID := idOffset;
IF enable THEN
	
	//wait(IN := errNo > 0, PT := T#1S);
	//IF wait.Q THEN
		errID := idOffset + errNo;
	//END_IF

END_IF

END_FUNCTION_BLOCK

// ---- POUs/MainPous/FC4_TpKommunikation/F_SAFETY_AnzeigenHohePrio.TcPOU
FUNCTION F_SAFETY_AnzeigenHohePrio : BOOL (* Ehemals F_PNOZ_AnzeigenHohePrio() *)
VAR_INPUT
END_VAR
VAR
END_VAR

(*    
	  U     "T 72"
      SPB   POK
*)
IF GVL.tonSAFETYok.Q THEN //(ehem. T72)
	RETURN;
END_IF


(*
      L     27  //PNOZ-Signal ungültig
      T     "DB6".w226_Betr_Anz_Wert
*)
DB6.w226_Betr_Anz_Wert := 127;

(*
      L     "DB6".w230
      L     24
      ==I   
      SPBN  a01
*)
IF (* DB6.w230 = 24 *) NOT IO.safeOutHauptLuft THEN
	(*
	 L    1                           //Druckluft nicht ein (weiter mit Masch-Ein)
	 T     "DB6".w226_Betr_Anz_Wert
	*)
	DB6.w226_Betr_Anz_Wert := 101;
END_IF
(*	  
a01:  BLD   130
      L     "DB6".w230
      L     48
      ==I   
      SPBN  a02
*)
IF (* DB6.w230 = 48 *) NOT IO.safeOutHauptLuft AND NOT IO.safeOutSchutzTueren THEN
	(*
	L     2   //Schutztür nicht zu
    T     "DB6".w226_Betr_Anz_Wert
	*)
	DB6.w226_Betr_Anz_Wert := 102;
END_IF
(*	  
      
a02:  BLD   130
      L     "DB6".w230
      L     68
      ==I   
      SPBN  a05
*)
IF (* DB6.w230 = 68 *) NOT IO.inResetNotHalt THEN
	(*
	L     5  //Kein Signal von Taste Maschine-Aus
    T     "DB6".w226_Betr_Anz_Wert
	*)
	DB6.w226_Betr_Anz_Wert := 105;
END_IF
(*	  
a05:  BLD   130
      L     "DB6".w230
      L     72
      ==I   
      SPBN  a08
*)
IF (* DB6.w230 = 72 *) NOT IO.safeOutHauptLuft AND NOT IO.safeOutNotHalt THEN
	(*
	 L     8                           //Not-Aus Steuerpult nicht OK     
     T     "DB6".w226_Betr_Anz_Wert
	*)
	DB6.w226_Betr_Anz_Wert := 108;
END_IF




(*	  
a08:  BLD   130
      U     "T 70"
      SPBN  a09
*)


//IF NOT GVL.tonPnozEntprell.Q THEN
//	RETURN;
//END_IF
(*
      L     9                           //Kein Signal von PNOZ
      T     "DB6".w226_Betr_Anz_Wert
*)
//DB6.w226_Betr_Anz_Wert := 109;
(*
a09:  BLD   130
POK:  BLD   130
*)

END_FUNCTION

// ---- POUs/MainPous/FC4_TpKommunikation/F_SignaldauerVonTastleuchte_MaschEinAuswerten.TcPOU
FUNCTION F_SignaldauerVonTastleuchte_MaschEinAuswerten : BOOL
VAR_INPUT
END_VAR
VAR
	wTmp : UDINT;
	setPnozSigLen : BOOL := FALSE;
END_VAR

//HIER WEITER
(*      
	  U     "E0_1"
      X     "M 3.1"
      SPBN  s1
*)

setPnozSigLen := FALSE;

IF IO.inResetNotHalt XOR VAT.bResetNotHalt_Old THEN //war M3.1

(*
      U     "E0_1"
      =     "M 3.1"
      SPB   zm
	  *)
	  //VAT.bResetNotHalt_Old := IO.inResetNotHalt; NBT - hier weggenommen...
	  //IF NOT IO.inResetNotHalt THEN
		  (*
		  L     999
		  L     "T 71"	-- gehe davon aus, dass er die Zeit von T71 lädt...
		  -I    		-- AKKU1 von AKKU2 subtrahieren
		  +     -1		-- Ganzzahl addieren
		  L     4
		  /I    		-- AKKU2 durch AKKU1 dividieren
		  L     4		
		  *I    		-- AKKU1 und AKKU2 multiplizieren
		  T     "DB6".w230
		  *)
		  //ToDo, noch keine Ahnung, was das soll...(LSB's verschwinden lassen)
		  //DB6.w230 := 999 - TIME_TO_INT(GVL.tofPnozSigLen.ET);
	  //END_IF
	  (*
zm:   BLD   130
      SET  -- VKE auf 1 setzen (=1)  
      L     S5T#9S990MS
      SA    "T 71" -- Zeit mit Ausschaltverzögerung start vorbereiten mit VKE=1
      CLR   VKE auf 0 setzen 
      SA    "T 71" -- Zeit mit Ausschaltverzögerung starten mit VKE=0
*)
setPnozSigLen := TRUE;
	  
END_IF //of IF IO.e01PNOZ_Signal XOR VAT.M3.1 ...

//GVL.tofPnozSigLen(IN := setPnozSigLen, PT := T#9S990MS); //(ehem. T71)

VAT.bResetNotHalt_Old := IO.inResetNotHalt; //NBT - hier hingesetzt...

(*	  
s1:   BLD   130
      UN    "E0_1"
      L     S5T#1S200MS
      SE    "T 70"
*)
//GVL.tonPnozEntprell(IN := NOT IO.inResetNotHalt, PT := T#1S200MS); //(ehem. T70)
(*	  
      U     "E0_1"
      L     S5T#1S
      SE    "T 72"
*)
//GVL.tonSAFETYok(IN := IO.safeOutHauptLuft, PT := T#1S); -- von hier weg nach P_InputHandling()

END_FUNCTION

// ---- POUs/MainPous/FC99_LetzterFC/P_LetzterFC.TcPOU
PROGRAM P_LetzterFC
VAR
END_VAR

(* Netzwerk: 1 *)
(*
TMD 40
TDB6.DBD 60
*)

(*
U "M0.2" M0.2 -- 2te Ablauf-Freigabe
= A 0.4
U "M 3.0" M3.0 -- Alles in Sollposition
= A 0.5
*)

//physische Ausgänge eintragen...
// A0.4 := VAT0.M0.2;
// A0.5 := VAT0.M0.3;

(* Netzwerk: 2 *)

(*
BEA -- Bausteinende absolut !!! ??? !!! Nur Test ?
U "E1_4" E1.4 -- R Abisolierer rück (abisoliert)
= A 0.4
NOT
= A 0.5
U "E1_5" E1.5 -- R Abisolierer links (aus Arbeitsraum)
= "A 0.6" A0.6 -- Y-1 Ausstoßen
NOT
= "A 0.7" A0.7 -- Y-2 Kontakt-Vereinzelung
*)

END_PROGRAM

// ---- GlobalTextList.TcGTLO
TEXTLIST GlobalTextList
  910 = '   E1.10 Kontakt gefallen' | EN: '   E1.10 Contact fallen' | DE: '   E1.10 Kontakt gefallen' | FR: '   E1.10 Contact tombé' | HU: '   E1.10 Érintkezo leesett' | IT: '   E1.10 Contatti caduti' | RU: '   E1.10 Контакт отсутствует' | RO: '   E1.10 Contact cazut' | ES: '   E1.10 Contacto caído' | PL: '   E1.10 Wypadnięcie kontaktu' | JA: '   E1.10 コンタクト脱落' | ZH: '   E1.10 针已落下'
  724 = '   E1.11 Crimpeinheit vorn' | EN: '   E1.11 Crimping unit at front' | DE: '   E1.11 Crimpeinheit vorn' | FR: '   E1.11 Unité de sertissage avance' | HU: '   E1.11 Krimpelo egység elöl' | IT: '   E1.11 Unità di crimpatura posizionata di fronte' | RU: '   E1.11 Передняя обжимная матрица' | RO: '   E1.11 Unitate de sertizare in fata' | ES: '   E1.11 Unidad de engaste en parte frontal' | PL: '   E1.11 Jednostka zaciskająca z przodu' | JA: '   E1.11 圧着ユニットが前面にあります' | ZH: '   E1.11 压接单元在前'
  875 = '   E1.12 Crimpeinheit rück' | EN: '   E1.12 Crimping unit at rear' | DE: '   E1.12 Crimpeinheit rück' | FR: '   E1.12 Unité de sertissage retour' | HU: '   E1.12 Krimpelo egység hátul' | IT: '   E1.12 Unità di crimpatura posizionata dietro' | RU: '   E1.12 Обжимной блок на задней панели' | RO: '   E1.12 Unitatea de sertizare in spate' | ES: '   E1.12 Unidad de crimpado en la parte posterior' | PL: '   E1.12 Jednostka zaciskająca z tyłu' | JA: '   E1.12 圧着ユニットが後方にあります' | ZH: '   E1.12 压接单元在后'
  515 = '   E1.13 Ausstoßen vorn' | EN: '   E1.13 Ejector at front' | DE: '   E1.13 Ausstoßen vorn' | FR: '   E1.13 Ejection avant' | HU: '   E1.13 Kilökés elöl' | IT: '   E1.13 Espulsore posizionato di fronte' | RU: '   E1.13 Экстрактор на фронтальной стороне' | RO: '   E1.13 Ejectorul in fata' | ES: '   E1.13 Eyector al frente' | PL: '   E1.13 Wyrzutnik z przodu' | JA: '   E1.13 エジェクタが前面に有ります' | ZH: '   E1.13 弹射器在前'
  869 = '   E1.14 Kontakt schieben vorn' | EN: '   E1.14 Contact slides at front' | DE: '   E1.14 Kont.Schieben vorn' | FR: '   E1.14 Pousser contact avant' | HU: '   E1.14 Érintk. tolása elöl' | IT: '   E1.14 Slitta contatti posizionata di fronte' | RU: '   E1.14 Завести контакт с фронтальной стороны' | RO: '   E1.14 Impingatoarele de contacte in fata' | ES: '   E1.14 Pasador de contactos en parte frontal' | PL: '   E1.14 Zjeżdżalnia dla kontaktów z przodu' | JA: '   E1.14 コンタクトが前面に有ります' | ZH: '   E1.14 推针器在前'
  858 = '   E1.15 Magazin gefüllt' | EN: '   E1.15 Magazine filled up' | DE: '   E1.15 Magazin gefüllt' | FR: '   E1.15 Magasin rempli' | HU: '   E1.15 Tároló feltöltve' | IT: '   E1.15 Caricatore pieno' | RU: '   E1.15 Магазин заполнен' | RO: '   E1.15 Magazie plina' | ES: '   E1.15 Depósito llenado' | PL: '   E1.15 Magazynek wypełniony' | JA: '   E1.15 マガジンが一杯です' | ZH: '   E1.15 填满料箱'
  1057 = '   E1.2 Drahthalter offen' | EN: '   E1.2 Wire holder open' | DE: '   E1.2 Drahthalter offen' | FR: '   E1.2 Porte-fil ouvert' | HU: '   E1.2 Huzaltartó nyitva' | IT: '   E1.2 Dispositivo blocca-cavo aperto' | RU: '   E1.2 Открыть кабельный захват' | RO: '   E1.2 Suport fir deschis' | ES: '   E1.2 Soporte de cable abierto' | PL: '   E1.2 Uchwyt przewodu otwarty' | JA: '   E1.2 ケーブルフォルダーオープン' | ZH: '   E1.2 集线器打开'
  122 = '   E1.3 Auslöseschalter' | EN: '   E1.3 Cable trigger switch' | DE: '   E1.3 Auslöseschalter' | FR: '   E1.3 Déclencheur' | HU: '   E1.3 Kioldó kapcsoló' | IT: '   E1.3 Sensore di presenza cavo' | RU: '   E1.3 Тригерный переключатель' | RO: '   E1.3 Comutator declansare' | ES: '   E1.3 Interruptor de disparo de cable' | PL: '   E1.3 Przełącznik kablowy' | JA: '   E1.3 ケーブルトリガースイッチ' | ZH: '   E1.3  线缆触发开关'
  459 = '   E1.4 Abisolierer zu' | EN: '   E1.4 Stripping unit closed' | DE: '   E1.4 Abisolierer  zu' | FR: '   E1.4 Dénudeur fermé' | HU: '   E1.4 Csupaszító zárva' | IT: '   E1.4 Unità di spellatura chiusa' | RU: '   E1.4 Закрыть блок зачистки' | RO: '   E1.4 Dezizolator inchis' | ES: '   E1.4 Unidad de pelado cerrada' | PL: '   E1.4 Jednostka odizolowująca zamknięta' | JA: '   E1.4 ストリッピングユニットクローズ' | ZH: '   E1.4 剥线单元闭合 '
  687 = '   E1.5 Abisolierer vorn' | EN: '   E1.5 Stripping unit at front' | DE: '   E1.5 Abisolierer vorn' | FR: '   E1.5 Dénudeur avance' | HU: '   E1.5 Csupaszító elöl' | IT: '   E1.5 Unità di spellatura posizionata di fronte' | RU: '   E1.5 Фронтальный блок зачистки' | RO: '   E1.5 Dezizolator in fata' | ES: '   E1.5 Unidad de pelado al frente' | PL: '   E1.5 Jednostka odizolowująca z przodu' | JA: '   E1.5 ストリッピングユニットが前面に有ります' | ZH: '   E1.5 剥线单元在前'
  302 = '   E1.6 Abisolierer rück' | EN: '   E1.6 Stripping unit at rear' | DE: '   E1.6 Abisolierer rück' | FR: '   E1.6 Dénudeur retour' | HU: '   E1.6 Csupaszító vissza' | IT: '   E1.6 Unità di spellatura posizionata dietro' | RU: '   E1.6 Блок зачистки на задней панели' | RO: '   E1.6 Dezizolator in spate' | ES: '   E1.6 Unidad de pelado atrás' | PL: '   E1.6 Jednostka odizolowująca z tyłu' | JA: '   E1.6 ストリッピングユニットが後方に有ります' | ZH: '   E1.6 剥线单元在后'
  982 = '   E1.7 Abisolierer links' | EN: '   E1.7 Stripping unit on LH side' | DE: '   E1.7 Abisolierer links' | FR: '   E1.7 Dénudeur gauche' | HU: '   E1.7 Csupaszító balra' | IT: '   E1.7 Unità di spellatura sul lato LH' | RU: '   E1.7 Левый блок зачистки' | RO: '   E1.7 Dezizolator in stanga' | ES: '   E1.7 Unidad de pelado  en lado LH' | PL: '   E1.7 Jednostka odizolowująca po lewej stronie' | JA: '   E1.7 ストリッピングユニットがLH側に有ります' | ZH: '   E1.7 剥线单元在左边'
  887 = '   E1.8 CrimpZange zu' | EN: '   E1.8 Crimping tool closed' | DE: '   E1.8 Crimpzange zu' | FR: '   E1.8 Pince à sertir fermée' | HU: '   E1.8 Krimpelo fogó zárva' | IT: '   E1.8 Ganasce di crimpatura chiuse' | RU: '   E1.8 Обжимная матрица закрыта' | RO: '   E1.8 Cleste sertizare inchis' | ES: '   E1.8 Herramienta de engaste cerrada' | PL: '   E1.8 Jednostka zaciskająca zamknięta' | JA: '   E1.8 圧着ツールクローズ' | ZH: '   E1.8 压接工具闭合'
  317 = '   E1.9 CrimpZange offen' | EN: '   E1.9 Crimping tool open' | DE: '   E1.9 Crimpzange offen' | FR: '   E1.9 Pince à sertir ouverte' | HU: '   E1.9 Krimpelo fogó nyitva' | IT: '   E1.9 Ganasce di crimpatura aperte' | RU: '   E1.9 Обжимная матрица открыта' | RO: '   E1.9 Cleste sertizare deschis' | ES: '   E1.9 Herramienta de engaste abierta' | PL: '   E1.9 Jednostka zaciskająca otwarta' | JA: '   E1.9 圧着ツールオープン' | ZH: '   E1.9 压接工具打开'
  891 = ' DE 1.10 Kontakt ist gefallen' | EN: '  DI 1.10 Contact fallen' | DE: ' DE 1.10 Kontakt gefallen' | FR: '  DI1.10 Contact tombé' | HU: '  DI1.10 Érintkezo leesett' | IT: '  DI1.10 Contatti caduti' | RU: '  DI1.10 Контакт отсутствует' | RO: '  DI1.10 Contact cazut' | ES: '  DI1.10 Contacto caído' | PL: '  DI1.10 Wypadnięcie kontaktu' | JA: '  DI1.10 コンタクト脱落' | ZH: '  DI1.10 针已落下'
  583 = ' DE 1.11 Crimpeinheit ist VORN' | EN: '  DI 1.11 Crimping unit at front' | DE: ' DE 1.11 Crimpeinheit vorn' | FR: '  DI1.11 Unité de sertissage avance' | HU: '  DI1.11 Krimpelo egység elöl' | IT: '  DI1.11 Unità di crimpatura posizionata di fronte' | RU: '  DI1.11 Передняя обжимная матрица' | RO: '  DI1.11 Unitate de sertizare in fata' | ES: '  DI1.11 Unidad de engaste en parte frontal' | PL: '  DI1.11 Jednostka zaciskająca z przodu' | JA: '  DI1.11 圧着ユニットが前面にあります' | ZH: '  DI1.11 压接单元在前'
  723 = ' DE 1.12 Crimpeinheit ist RUECK\t' | EN: '  DI 1.12 Crimping unit at rear' | DE: ' DE 1.12 Crimpeinheit rück' | FR: '  DI1.12 Unité de sertissage retour' | HU: '  DI1.12 Krimpelo egység hátul' | IT: '  DI1.12 Unità di crimpatura posizionata dietro' | RU: '  DI1.12 Обжимной блок на задней панели' | RO: '  DI1.12 Unitatea de sertizare in spate' | ES: '  DI1.12 Unidad de crimpado en la parte posterior' | PL: '  DI1.12 Jednostka zaciskająca z tyłu' | JA: '  DI1.12 圧着ユニットが後方にあります' | ZH: '  DI1.12 压接单元在后'
  285 = ' DE 1.13 Ausstossen VORN' | EN: '  DI 1.13 Ejector at front' | DE: ' DE 1.13 Ausstoßen vorn' | FR: '  DI1.13 Ejection avant' | HU: '  DI1.13 Kilökés elöl' | IT: '  DI1.13 Espulsore posizionato di fronte' | RU: '  DI1.13 Экстрактор на фронтальной стороне' | RO: '  DI1.13 Ejectorul in fata' | ES: '  DI1.13 Eyector al frente' | PL: '  DI1.13 Wyrzutnik z przodu' | JA: '  DI1.13 エジェクタが前面に有ります' | ZH: '  DI1.13 弹射器在前'
  650 = ' DE 1.14 Kontakt schieben VORN' | EN: '  DI 1.14 Contact slides at front' | DE: ' DE 1.14 Kont.Schieben vorn' | FR: '  DI1.14 Pousser contact avant' | HU: '  DI1.14 Érintk. tolása elöl' | IT: '  DI1.14  Slitta contatti posizionata di fronte' | RU: '  DI1.14 Завести контакт с фронтальной стороны' | RO: '  DI1.14 Impingatoarele de contacte in fata' | ES: '  DI1.14 Pasador de contactos en parte frontal' | PL: '  DI1.14 Zjeżdżalnia dla kontaktów z przodu' | JA: '  DI1.14 コンタクトが前面に有ります' | ZH: '  DI1.14 推针器在前'
  752 = ' DE 1.15 Magazin GEFÜLLT' | EN: '  DI 1.15 Magazine filled up' | DE: ' DE 1.15 Magazin gefüllt' | FR: '  DI1.15 Magasin rempli' | HU: '  DI1.15 Tároló feltöltve' | IT: '  DI1.15 Caricatore pieno' | RU: '  DI1.15 Магазин заполнен' | RO: '  DI1.15 Magazie plina' | ES: '  DI1.15 Depósito llenado' | PL: '  DI1.15 Magazynek wypełniony' | JA: '  DI1.15 マガジンが一杯です' | ZH: '  DI1.15 填满料箱'
  819 = ' DE 1.2 Drahthalter ist Offen' | EN: '  DI 1.2 Wire holder open' | DE: ' DE 1.2 Drahthalter offen' | FR: '  DI1.2 Porte-fil ouvert' | HU: '  DI1.2 Huzaltartó nyitva' | IT: '  DI1.2 Dispositivo blocca-cavo aperto' | RU: '  DI1.2 Открыть кабельный захват' | RO: '  DI1.2 Suport fir deschis' | ES: '  DI1.2 Soporte de cable abierto' | PL: '  DI1.2 Uchwyt przewodu otwarty' | JA: '  DI1.2 ケーブルフォルダーオープン' | ZH: '  DI1.2 集线器打开'
  771 = ' DE 1.3 Auslöse Schalter' | EN: '  DI 1.3 Cable trigger switch' | DE: ' DE 1.3 Auslöseschalter' | FR: '  DI1.3 Déclencheur' | HU: '  DI1.3 Kioldó kapcsoló' | IT: '  DI1.3 Sensore di presenza cavo' | RU: '  DI1.3 Тригерный переключатель' | RO: '  DI1.3 Comutator declansare' | ES: '  DI1.3 Interruptor de disparo de cable' | PL: '  DI1.3 Przełącznik kablowy' | JA: '  DI1.3 ケーブルトリガースイッチ' | ZH: '  DI1.3  线缆触发开关'
  256 = ' DE 1.4 Abisolierer ist ZU\t' | EN: '  DI 1.4 Stripping unit closed' | DE: ' DE 1.4 Abisolierer  zu' | FR: '  DI1.4 Dénudeur fermé' | HU: '  DI1.4 Csupaszító zárva' | IT: '  DI1.4 Unità di spellatura chiusa' | RU: '  DI1.4 Закрыть блок зачистки' | RO: '  DI1.4 Dezizolator inchis' | ES: '  DI1.4 Unidad de pelado cerrada' | PL: '  DI1.4 Jednostka odizolowująca zamknięta' | JA: '  DI1.4 ストリッピングユニットクローズ' | ZH: '  DI1.4 剥线单元闭合 '
  591 = ' DE 1.5 Abisolierer ist VORN' | EN: '  DI 1.5 Stripping unit at front' | DE: ' DE 1.5 Abisolierer vorn' | FR: '  DI1.5 Dénudeur avance' | HU: '  DI1.5 Csupaszító elöl' | IT: '  DI1.5 Unità di spellatura posizionata di fronte' | RU: '  DI1.5 Фронтальный блок зачистки' | RO: '  DI1.5 Dezizolator in fata' | ES: '  DI1.5 Unidad de pelado al frente' | PL: '  DI1.5 Jednostka odizolowująca z przodu' | JA: '  DI1.5 ストリッピングユニットが前面に有ります' | ZH: '  DI1.5 剥线单元在前'
  315 = ' DE 1.6 Abisolierer ist RÜCK' | EN: '  DI 1.6 Stripping unit at rear' | DE: ' DE 1.6 Abisolierer rück' | FR: '  DI1.6 Dénudeur retour' | HU: '  DI1.6 Csupaszító vissza' | IT: '  DI1.6 Unità di spellatura posizionata dietro' | RU: '  DI1.6 Блок зачистки на задней панели' | RO: '  DI1.6 Dezizolator in spate' | ES: '  DI1.6 Unidad de pelado atrás' | PL: '  DI1.6 Jednostka odizolowująca z tyłu' | JA: '  DI1.6 ストリッピングユニットが後方に有ります' | ZH: '  DI1.6 剥线单元在后'
  227 = ' DE 1.7 Abisolierer ist LINKS' | EN: '  DI 1.7 Stripping unit on LH side' | DE: ' DE 1.7 Abisolierer links' | FR: '  DI1.7 Dénudeur gauche' | HU: '  DI1.7 Csupaszító balra' | IT: '  DI1.7 Unità di spellatura sul lato LH' | RU: '  DI1.7 Левый блок зачистки' | RO: '  DI1.7 Dezizolator in stanga' | ES: '  DI1.7 Unidad de pelado  en lado LH' | PL: '  DI1.7 Jednostka odizolowująca po lewej stronie' | JA: '  DI1.7 ストリッピングユニットがLH側に有ります' | ZH: '  DI1.7 剥线单元在左边'
  935 = ' DE 1.8 Crimpzange ist ZU' | EN: '  DI 1.8 Crimping tool closed' | DE: ' DE 1.8 Crimpzange zu' | FR: '  DI1.8 Pince à sertir fermée' | HU: '  DI1.8 Krimpelo fogó zárva' | IT: '  DI1.8 Ganasce di crimpatura chiuse' | RU: '  DI1.8 Обжимная матрица закрыта' | RO: '  DI1.8 Cleste sertizare inchis' | ES: '  DI1.8 Herramienta de engaste cerrada' | PL: '  DI1.8 Jednostka zaciskająca zamknięta' | JA: '  DI1.8 圧着ツールクローズ' | ZH: '  DI1.8 压接工具闭合'
  187 = ' DE 1.9 Crimpzange ist OFFEN' | EN: '  DI 1.9 Crimping tool open' | DE: ' DE 1.9 Crimpzange offen' | FR: '  DI1.9 Pince à sertir ouverte' | HU: '  DI1.9 Krimpelo fogó nyitva' | IT: '  DI1.9 Ganasce di crimpatura aperte' | RU: '  DI1.9 Обжимная матрица открыта' | RO: '  DI1.9 Cleste sertizare deschis' | ES: '  DI1.9 Herramienta de engaste abierta' | PL: '  DI1.9 Jednostka zaciskająca otwarta' | JA: '  DI1.9 圧着ツールオープン' | ZH: '  DI1.9 压接工具打开'
  448 = '%0.1f bar' | EN: '%0.1f bars' | DE: '%0.1f bar' | FR: '%0.1f bars' | HU: '%0.1f bar' | IT: '%0.1f bar' | RU: '%0.1f бар' | RO: '%0.1f bar' | ES: '%0.1f bar' | PL: '%0.1f bar' | JA: '%0.1f bar' | ZH: '%0.1f bar'
  513 = '%0.1f Sek' | EN: '%0.1f sec' | DE: '%0.1f Sek' | FR: '%0.1f sec' | HU: '%0.1f sec' | IT: '%0.1f sec' | RU: '%0.1f сек' | RO: '%0.1f sec' | ES: '%0.1f sec' | PL: '%0.1f sec' | JA: '%0.1f sec' | ZH: '%0.1f sec'
  44 = '%d' | EN: '%d' | DE: '%d' | FR: '%d' | HU: '%d' | IT: '%d' | RU: '%d' | RO: '%d' | ES: '%d' | PL: '%d' | JA: '%d' | ZH: '%d'
  60 = '%s' | EN: '%s' | DE: '%s' | FR: '%s' | HU: '%s' | IT: '%s' | RU: '%s' | RO: '%s' | ES: '%s' | PL: '%s' | JA: '%s' | ZH: '%s'
  707 = 'A1.10-AbisoliererLINKS' | EN: 'A1.10-Stripping unit to LH side' | DE: 'A1.10-Abisolierer links' | FR: 'A1.10-Dénudeur gauche' | HU: 'A1.10-Csupaszító balra' | IT: 'A1.10-Unità di spellatura sul lato LH' | RU: 'A1.10-Левый блок зачистки' | RO: 'A1.10-Dezizolator in stanga' | ES: 'A1.10-Unidad de pelado  en lado LH' | PL: 'A1.10-Jednostka odizolowująca po lewej stronie' | JA: 'A1.10-ストリッピングユニットがLH側に有ります' | ZH: 'A1.10-剥线单元在左边'
  708 = 'A1.11-AbisoliererZU' | EN: 'A1.11-CLOSE StrippingUnit' | DE: 'A1.11-Abisolierer  zu' | FR: 'A1.11-Dénudeur fermé' | HU: 'A1.11-Csupaszító zárva' | IT: 'A1.11-Unità di spellatura chiusa' | RU: 'A1.11-Закрыть блок зачистки' | RO: 'A1.11-Dezizolator inchis' | ES: 'A1.11-Unidad de pelado cerrada' | PL: 'A1.11-Jednostka odizolowująca zamknięta' | JA: 'A1.11-ストリッピングユニットクローズ' | ZH: 'A1.11-剥线单元闭合 '
  64 = 'A1.12-AbfallRUNTER' | EN: 'A1.12-Waste DOWN' | DE: 'A1.12-AbfallRUNTER' | FR: 'A1.12-Déchets en aval'
  709 = 'A1.13-AbisoliererRUECK' | EN: 'A1.13-StrippingUnit to REAR' | DE: 'A1.13-AbisoliererRUECK'
  710 = 'A1.14-CrimperZU' | EN: 'A1.14-CLOSE CrimpingTool' | DE: 'A1.14-CrimperZU'
  62 = 'A1.15-DrahthaltFüh.ZU' | EN: 'A1.15-CLOSE WireHolder' | DE: 'A1.15-DrahthaltFüh.ZU'
  703 = 'A1.5-Sortierluft' | EN: 'A1.5-Sorting Air ON' | DE: 'A1.5-Sortierluft'
  704 = 'A1.6-Ausstossen' | EN: 'A1.6-Ejector to FRONT' | DE: 'A1.6-Ausstossen'
  705 = 'A1.7-KontaktVereinz.' | EN: 'A1.8-Contact separating ON' | DE: 'A1.7-KontaktVereinz.'
  63 = 'A1.8-KontaktSchieben' | EN: 'A1.8-SLIDE Contact' | DE: 'A1.8-KontaktSchieben'
  706 = 'A1.9-CrimpEinheitVOR' | EN: 'A1.9-CrimpingTool to FRONT' | DE: 'A1.9-CrimpEinheitVOR'
  874 = 'Abisolierung einrichten' | EN: 'Set up stripping unit' | DE: 'Abisolierung einrichten' | FR: 'Réglage dénudage' | HU: 'Csupaszítás beállítása' | IT: 'Regolazione unità di spellatura' | RU: 'Настройка снятия изоляции' | RO: 'Reglare dezizolare' | ES: 'Configurar unidad de pelado' | PL: 'Ustawianie jednostki odizolowującej' | JA: 'ストリッピング・ユニットをセットしてください' | ZH: '设置剥线单元'
  638 = 'AUF' | EN: 'OPEN' | DE: 'AUF' | FR: 'OUVERT' | HU: 'Nyit' | IT: 'Aperto' | RU: 'Открыть' | RO: 'Deschide' | ES: 'Abierto' | PL: 'Otwórz' | JA: '開く' | ZH: '打开'
  702 = 'Ausgangs-Test' | EN: 'Output-Test' | DE: 'Ausgangs-Test'
  386 = 'Auslösesch.:' | EN: 'Trigger switch.:' | DE: 'Auslösesch.:' | FR: 'Déclencheur:' | HU: 'Kioldó kapcsoló:' | IT: 'Sens.di cavo:' | RU: 'Переключатель:' | RO: 'Comutator dec.:' | ES: 'Inter.de de cable:' | PL: 'Przełącznik:' | JA: 'ケーブルトリガースイッチ' | ZH: '线缆触发开关'
  42 = 'Ausstoßverzögerung' | EN: 'Discharge delay' | DE: 'Ausstoßverzögerung' | FR: "Retardement d'éjection" | HU: 'Kidobási késleltetés' | IT: 'Ritardo di espulsione' | RU: 'Задержка выталкивания' | RO: 'Intarziere ejectare' | ES: 'Retardo de descarga' | PL: 'Opóźnienie wydawania' | JA: 'イジェクト時間' | ZH: '弹出时间'
  233 = 'Ausstoßzeit' | EN: 'Ejection time' | DE: 'Ausstoßzeit' | FR: "Durée d'éjection" | HU: 'Kidobási ido' | IT: 'Tempo di espulsione' | RU: 'Время выталкивания' | RO: 'Timp de ejectie' | ES: 'Tiempo de eyección' | PL: 'Czas wyrzutu' | JA: '駆出遅延' | ZH: '弹出延迟'
  524 = 'Bei kleinen Kontakten mit labiler Litze, muss diese unmittelbar nach dem Crimpen von Hand herausgezogen werden. Dazu kann hier eine Verzögerungszeit eingegeben werden. (Wert 0 = ohne Verzögerung)' | EN: 'In the case of smaller contacts with fragile wire, it is necessary to manually pull it out immediately after crimping. A delay time can be entered for this step. (Value 0 = without delay)' | DE: 'Bei kleinen Kontakten mit labiler Litze, muss diese unmittelbar nach dem Crimpen von Hand herausgezogen werden. Dazu kann hier eine Verzögerungszeit eingegeben werden. (Wert 0 = ohne Verzögerung)' | FR: 'En cas de petits contacts avec des lithes instables, ceux-ci doivent être retirés à la main immédiatement après le crimpage. Pour ce faire, un délai de retard peut être saisi ici. (valeur 0 = sans délai)' | HU: 'Ha kis érintkezok huzala labilis, akkor közvetlenül a krimpelés után ki kell húzni azt.\nEhhez be lehet írni késleltetési idot. (0 érték = nincs késleltetési ido)' | IT: "Nel caso di cavi di piccola sezione, è necessario aiutare manualmente l'espulsione del cavo crimpato tirando il cavo stesso verso l'esterno alla fine dell'operazione di crimpatura. E' possibile impostare un ritardo per questa operazione (valore 0 = NO ritardo)" | RU: 'В случае контактов под кабель небольшого сечения, извлечь сразу же вручную после обжима.\nДля этого задается время задержки. (Значение 0 = без задержки)' | RO: 'La contactele mici, cu fir labil, aceasta trebuie indepărtata manual imediat după sertizare.\nDin acest motiv se poate introduce aici un timp de întârziere. (Valoare 0 = nici o întârziere)' | ES: 'En el caso de los contactos para secciones más pequeñas, es necesario extraerlos después del engaste. \nUn tiempo de retardo puede ser ajustado para este paso. (Valor 0 = sin retardo)' | PL: 'W przypadku małych kontaktów z delikatnymi przewodami, konieczne jest manualne wyciągnięcie natychmiast po zacisku.\nCzas opóźnienia może być wprowadzony dla tego kroku (Wartość 0 = bez opóźnienia)' | JA: '細いコンタクトで柔らかいケーブルを圧着する場合、機械がコンタクトを圧着したタイミングで速やかにコンタクトを引き出してください\u3000タイミング調整はこのステップで調整できます（値0＝遅れなし' | ZH: '当细针压接很细的线,需要在压接之后立刻手动将针拉出来.在这个操作可以设定一定的延迟时间. (值为 0 = 没有延迟)'
  886 = 'BetrAnz.: %d'
  286 = 'Betriebsstunden:' | EN: 'Operating hours' | DE: 'Betriebsstunden' | FR: 'Pour des petits contacts avec un fil instable, retirer à la main immédiatement à la suite du sertissage. Pour cela, il est possible de saisir un temps de retardement. (Valeur 0 = sans retardement)' | HU: 'Üzemórák' | IT: 'Ore di lavoro' | RU: 'Эксплуатационное время' | RO: 'Ore functionare' | ES: 'Horas de operación' | PL: 'Ilość godzin pracy' | JA: '作業時間' | ZH: '运行时间'
  1124 = 'c'
  964 = 'Chinesisch' | EN: 'Chinese' | DE: 'Chinesisch' | FR: 'Chinois' | HU: 'Kínai' | IT: 'Cinese' | RU: 'китайский' | RO: 'chineză' | ES: 'Chino' | PL: 'Chiński' | JA: '中国の' | ZH: '中国'
  876 = 'Crimpen' | EN: 'Crimping' | DE: 'Crimpen' | FR: 'Sertir' | HU: 'Krimpelés' | IT: 'Crimpatura' | RU: 'Обжим' | RO: 'Sertizare' | ES: 'Engastando' | PL: 'Zaciskanie' | JA: '圧着' | ZH: '压接'
  817 = 'Crimpzange einrichten' | EN: 'Set up crimping tool' | DE: 'Crimpzange einrichten' | FR: 'Réglage pince de sertissage' | HU: 'Krimpelo fogó beállítása' | IT: 'Regolazione unità di crimpatura' | RU: 'Настройка обжимного элемента' | RO: 'Reglare cleste sertizare' | ES: 'Ajuste herramienta de engastado' | PL: 'Ustawianie jednostki zaciskającej' | JA: '圧着ツールのセットアップ' | ZH: '设定压接工具'
  372 = 'DE Klemme EL1809-01'
  973 = 'DE Klemme EL1809-02'
  581 = 'Deutsch' | EN: 'German' | DE: 'Deutsch' | FR: 'Allemand' | HU: 'Német' | IT: 'Tedesco' | RU: 'Немецкий' | RO: 'Germana' | ES: 'Alemán' | PL: 'Niemiecki' | JA: 'ドイツ語' | ZH: '德语'
  740 = 'Drahthalter Druck' | EN: 'Wire holder pressure' | DE: 'Drahthalter Druck' | FR: 'Pression de support de fil' | HU: 'Huzal tartó nyomása' | IT: 'Pressione del supporto del filo' | RU: 'Давление в держателе' | RO: 'Presiunea suportului de susținere' | ES: 'Presión del soporte de alambre' | PL: 'Nacisk uchwytu drutu' | JA: 'ワイヤーホルダーの圧力' | ZH: '集线器压力'
  551 = 'Drahthalter:' | EN: 'wire holder' | DE: 'Drahthalter' | FR: 'support de fil' | HU: 'drótra' | IT: 'supporto del legare' | RU: 'держатель провода' | RO: 'titularul de sârmă' | ES: 'soporte de alambre' | PL: 'uchwyt na drut' | JA: '電線ホルダー' | ZH: '集线器'
  30 = 'Einzel/Auto' | EN: 'Single / Auto' | DE: 'Einzel/Auto' | FR: 'Simple / Auto' | HU: 'Single / Auto' | IT: 'Singolo / Auto' | RU: 'Одном./Aвто' | RO: 'Single / Auto' | ES: 'Individual / Auto' | PL: 'Single / Auto' | JA: 'シングル/オート' | ZH: '单个/自动'
  91 = 'Englisch' | EN: 'English' | DE: 'Englisch' | FR: 'Anglais' | HU: 'Angol' | IT: 'Inglese' | RU: 'Английский' | RO: 'Engleză' | ES: 'Inglés' | PL: 'Angielski' | JA: '英語' | ZH: '英文'
  730 = 'Ergebnis' | EN: 'Result' | DE: 'Ergebnis'
  640 = 'Esc' | EN: 'Esc' | DE: 'Esc' | FR: 'Esc' | HU: 'Esc' | IT: 'Esc' | RU: 'Esc' | RO: 'Esc' | ES: 'Esc' | PL: 'Esc' | JA: 'Esc' | ZH: '退出'
  214 = 'Fertig:' | EN: 'Finished' | DE: 'Fertig' | FR: 'Fini' | HU: 'Kész' | IT: 'Crimpature effettuate' | RU: 'Готово' | RO: 'Incheiat' | ES: 'Finalizado' | PL: 'Skończone' | JA: '終了' | ZH: '完成'
  714 = 'Französisch' | EN: 'French' | DE: 'Französisch' | FR: 'Français' | HU: 'Francia' | IT: 'Francese' | RU: 'Францу́зский' | RO: 'Franceză' | ES: 'Francés' | PL: 'Francuski' | JA: 'フランス語' | ZH: '法国'
  761 = 'HARTING Crimpautomat TK-M' | EN: 'HARTING Crimping Machine TK-M' | DE: 'HARTING Crimpautomat TK-M' | FR: 'Automate de sertissage TK-M HARTING' | HU: 'HARTING TK-M automata krimpelo gép' | IT: 'Crimpatrice HARTING TK-M' | RU: 'HARTING обжимная машина TK-M' | RO: 'Automat sertizare HARTING TK-M' | ES: 'Máquina de engaste TK-M de HARTING' | PL: 'HARTING maszyna zaciskająca TK-M' | JA: 'ハーティング自動圧着機\u3000TK-M' | ZH: 'HARTING 自动压接机 TK-M'
  311 = 'Italienisch' | EN: 'Italian' | DE: 'Italienisch' | FR: 'Italien' | HU: 'Olasz' | IT: 'Italiano' | RU: 'Италья́нский' | RO: 'Italiană' | ES: 'Italiano' | PL: 'Włoski' | JA: 'イタリア語' | ZH: '意大利'
  993 = 'Japanisch' | EN: 'Japanese' | DE: 'Japanisch' | FR: 'Japonais' | HU: 'Japán' | IT: 'Giapponese' | RU: 'японский' | RO: 'Japoneză' | ES: 'Japonés' | PL: 'Japoński' | JA: '日本の' | ZH: '日本'
  110 = 'Löschen' | EN: 'Delete' | DE: 'Löschen' | FR: 'Effacer' | HU: 'Törlés' | IT: 'Cancella' | RU: 'Удалить' | RO: 'Sterge' | ES: 'Borrar' | PL: 'Kasowanie' | JA: '削除' | ZH: '删除'
  816 = 'Magazin leerfahren' | EN: 'Run magazine empty' | DE: 'Magazin leerfahren' | FR: 'Vider le magasin' | HU: 'Tároló üresre járatása' | IT: 'Scarico canale contatti' | RU: 'Очистить магазин' | RO: 'Golire magazie' | ES: 'Ejecutar vaciado de depósito' | PL: 'Uruchom magazynek pusty' | JA: 'マガジンを空にする' | ZH: '运行料箱清空'
  355 = 'Menü' | EN: 'Menu' | DE: 'Menü' | FR: 'Menu' | HU: 'Menü' | IT: 'Menù' | RU: 'Меню' | RO: 'Meniu' | ES: 'Menu' | PL: 'Menu' | JA: 'メニュー' | ZH: '操作菜单'
  429 = 'Noch: %d' | EN: 'Still: %d' | DE: 'Noch: %d' | FR: 'Encore:  %d' | HU: 'Még:  %d' | IT: 'Mancanti:' | RU: 'Eще:  %d' | RO: 'Inca:  %d' | ES: 'Todavía:  %d' | PL: 'Wciąż:  %d' | JA: 'まだ:  %d' | ZH: '继续:  %d'
  919 = 'Off- / On Line'
  634 = 'Offline: Low / High'
  765 = 'ohne Sortierluft' | EN: 'without sorting air' | FR: "sans tri d'air" | HU: 'buborékok nélkül' | IT: 'senza aria' | RU: 'без пузырьков' | RO: 'fără bule' | ES: 'sin burbujas' | PL: 'bez bąbelków' | JA: '空気をソートせずに' | ZH: '没有分拣气'
  527 = 'OutTest'
  514 = 'Polnisch' | EN: 'Polish' | DE: 'Polnisch' | FR: 'Polonais' | HU: 'Lengyel' | IT: 'Polacco' | RU: 'Польский' | RO: 'Polonez' | ES: 'Polaco' | PL: 'Polski' | JA: 'ポーランド語' | ZH: '波兰语'
  590 = 'Probelauf' | EN: 'Trial run' | DE: 'Probelauf' | FR: "Marche d'essai" | HU: 'Próbaüzem' | IT: 'Ciclo di prova' | RU: 'Тест' | RO: 'Test' | ES: 'Modo de prueba' | PL: 'Przebieg testowy' | JA: 'テスト動作' | ZH: '试运行'
  92 = 'Probelauf ohne Crimpen' | EN: 'Trial run without crimping' | DE: 'Probelauf ohne Crimpen' | FR: "Marche d'essai sans sertissage" | HU: 'Próbaüzem krimpelés nélkül' | IT: 'Ciclo di prova senza crimpatura' | RU: 'Тест без обжима' | RO: 'Test fara sertizare' | ES: 'Prueba sin engaste' | PL: 'Przebieg testowy bez zaciskania' | JA: '圧着なしでのテスト動作' | ZH: '不压接试运行'
  371 = 'Probelauf ohne Kontakt' | EN: 'Trial run without contact' | DE: 'Probelauf ohne Kontakt' | FR: "Marche d'essai sans contact" | HU: 'Próbaüzem érintkezo nélkül' | IT: 'Ciclo di prova senza contatto' | RU: 'Тест без контакта' | RO: 'Test fara contact' | ES: 'Prueba sin contacto' | PL: 'Przebieg testowy bez kontaktu' | JA: 'コンタクトなしでのテスト動作' | ZH: '不带针试运行'
  61 = 'Probelauf ohne Litze' | EN: 'Trial run without wire' | DE: 'Probelauf ohne Litze' | FR: "Marche d'essai sans fil" | HU: 'Próbaüzem huzal nélkül' | IT: 'Ciclo di prova senza cavo' | RU: 'Тест без провода' | RO: 'Test fara lita' | ES: 'Prueba sin cable' | PL: 'Przebieg testowy bez przewodu' | JA: 'ケーブルなしでのテスト動作' | ZH: '不带线试运行'
  896 = 'R' | EN: 'R' | DE: 'R'
  786 = 'Reset' | EN: 'Reset' | DE: 'Reset' | FR: 'Reset' | HU: 'Visszaállítás' | IT: 'Reset' | RU: 'Перезагрузка' | RO: 'Reset' | ES: 'Reset' | PL: 'Reset' | JA: 'リセット' | ZH: '重置'
  770 = 'Rezeptur' | EN: 'Recipe' | DE: 'Rezeptur' | FR: 'Recette' | HU: 'Receptúra' | IT: 'Menù' | RU: 'Рецепт' | RO: 'Reteta' | ES: 'Receta' | PL: 'Przepis' | JA: 'レシピ' | ZH: '接收'
  339 = 'Rumänisch' | EN: 'Romanian' | DE: 'Rumänisch' | FR: 'Roumain' | HU: 'Román' | IT: 'Rumeno' | RU: 'Румы́нский' | RO: 'Român' | ES: 'Rumano' | PL: 'Rumuński' | JA: 'ルーマニア語' | ZH: '罗马尼亚'
  985 = 'Russisch' | EN: 'Russian' | DE: 'Russisch' | FR: 'Russe' | HU: 'Orosz' | IT: 'Russo' | RU: 'ру́сский' | RO: 'Rusă' | ES: 'Ruso' | PL: 'rosyjski' | JA: 'ロシア' | ZH: '俄'
  366 = 'Sensoren brücken' | EN: 'Sensor bridging' | DE: 'Sensoren brücken' | FR: 'Invalidation de capteurs' | HU: 'Érzékelok áthidalása' | IT: 'Disattivazione sensori' | RU: 'Шунтировать датчик' | RO: 'Ocolire senzor' | ES: 'Puenteo del sensor' | PL: 'Mostkowanie czujników' | JA: 'センサーブリッジ' | ZH: '传感器桥接'
  503 = 'Sensoren Brücken'
  790 = 'Sortierer leerfahren' | EN: 'Run sorter empty' | DE: 'Sortierer leerfahren' | FR: 'Vider trieuse' | HU: 'Szortírozó üresre járatása' | IT: 'Svuotamento contenitore contatti' | RU: 'Холостой ход сортировщика' | RO: 'Golire sortator' | ES: 'Ejecutar vaciado de clasificador' | PL: 'Uruchom sorter pusty' | JA: 'ソーター空ので動作' | ZH: '运行分拣清空'
  313 = 'Sortierer:' | EN: 'Sorter:' | DE: 'Sortierer:' | FR: 'Trieuse :' | HU: 'Szortírozó berendezés:' | IT: 'Livello vibrazione' | RU: 'Сортировщик:' | RO: 'Sortator:' | ES: 'Clasificador:' | PL: 'Sorter:' | JA: 'ソーター' | ZH: '分拣:'
  901 = 'Spanisch' | EN: 'Spanish' | DE: 'Spanisch' | FR: 'Espagnol' | HU: 'Spanyol' | IT: 'Spagnolo' | RU: 'Испа́нский' | RO: 'Spaniolă' | ES: 'Español' | PL: 'Hiszpański' | JA: 'スペイン語' | ZH: '西班牙语'
  840 = 'Speichern' | EN: 'Save' | DE: 'Speichern' | FR: 'Enregistrer' | HU: 'Mentés' | IT: 'Salvare' | RU: 'Сохранить' | RO: 'Salveaza' | ES: 'Guardar' | PL: 'Zapisz' | JA: '保存' | ZH: '保存'
  217 = 'Sprache' | EN: 'Language' | DE: 'Sprache' | FR: 'Langue' | HU: 'Nyelv' | IT: 'Lingua' | RU: 'Язык' | RO: 'Limba' | ES: 'Idioma' | PL: 'Język' | JA: '言語' | ZH: '语言'
  543 = 'Status' | EN: 'Status' | DE: 'Status' | FR: 'Statut' | HU: 'Állapot' | IT: 'Status' | RU: 'Статус' | RO: 'Stadiu' | ES: 'Estado' | PL: 'Status' | JA: '状態' | ZH: '状态'
  382 = 'Stop' | EN: 'Stop' | DE: 'Stop' | FR: 'Stop' | HU: 'Leállítás' | IT: 'Stop' | RU: 'Стоп' | RO: 'Stop' | ES: 'Parada' | PL: 'Stop' | JA: '停止' | ZH: '停止'
  486 = 'Stückzahl-Total:' | EN: 'Total quantity' | DE: 'Stückzahl Total' | FR: 'Nombre de pièces total' | HU: 'Összes darabszám' | IT: 'Contatore parziale' | RU: 'Общее кол-во' | RO: 'Cantitate totala' | ES: 'Cantidad total' | PL: 'Ilość całkowita' | JA: '設定数量' | ZH: '总数'
  949 = 'Stückzahl-Vorwahl' | EN: 'Quantity presel.' | DE: 'Stückzahl-Vorwahl' | FR: 'Présélection nombre de pièces' | HU: 'Darabszám eloválasztása' | IT: 'Impostazione quantità crimpature' | RU: 'Выбор кол-ва' | RO: 'Preselectie cantitate' | ES: 'Cantidad preseleccionada' | PL: 'Ilość wybór wstępny' | JA: 'トータル数量' | ZH: '预设总数.'
  332 = 'System'
  269 = 'Tageszähler:' | EN: 'Daily counter:' | DE: 'Tageszähler:' | FR: 'Compteur journalier :' | HU: 'Napi számláló:' | IT: 'Contatore giornaliero' | RU: 'Дневной счетчик' | RO: 'Numarator zilnic:' | ES: 'Contador diario:' | PL: 'Licznik dzienny:' | JA: 'デイリーカウンター' | ZH: '每日计数:'
  234 = 'Totalzähler' | EN: 'Total counter' | DE: 'Totalzähler' | FR: 'Compteur total' | HU: 'Összes számláló' | IT: 'Contatore totale' | RU: 'Общий счетчик' | RO: 'Numarator total' | ES: 'Contador total:' | PL: 'Licznik całkowity' | JA: 'トータルカウンター' | ZH: '总数'
  1113 = 'Um Abdrücke des Drahthalters auf dem Isoliermantel zu vermeiden, kann hier der Pneumatik-Druck des Drahthalters zwischen 0,5 und 6,0 bar eingestellt werden.' | EN: 'In order to avoid impressions of the wire holder on the insulating jacket, the pneumatic pressure of the wire holder can be adjusted here between 0.5 and 6.0 bar.' | DE: 'Um Abdrücke des Drahthalters auf dem Isoliermantel zu vermeiden, kann hier der Pneumatik-Druck des Drahthalters zwischen 0,5 und 6,0 bar eingestellt werden.' | FR: "Afin d'éviter les empreintes du porte-fil sur la chemise isolante, la pression pneumatique du porte-fil peut être ajustée ici entre 0,5 et 6,0 bars." | HU: 'Annak érdekében, hogy elkerülje a szigetelő burkolat dróttartójának benyomódását, a vezetéktartó pneumatikus nyomása 0,5 és 6,0 bar között állítható.' | IT: 'Al fine di evitare impronte del supporto del filo sulla guaina isolante, la pressione pneumatica del supporto del filo può essere regolata qui tra 0,5 e 6,0 bar.' | RU: 'Чтобы избежать впечатлений от держателя проволоки на изолирующем кожухе, пневматическое давление держателя проволоки можно регулировать здесь от 0,5 до 6,0 бар.' | RO: 'Pentru a evita impresiile suportului de sârmă de pe mantaua izolatoare, presiunea pneumatică a suportului de sârmă poate fi reglată aici între 0,5 și 6,0 bari.' | ES: 'Para evitar impresiones del soporte del cable en la camisa aislante, la presión neumática del soporte del cable se puede ajustar aquí entre 0,5 y 6,0 bar.' | PL: 'Aby uniknąć odcisków drutu na płaszczu izolacyjnym, ciśnienie pneumatyczne uchwytu drutu można ustawić w zakresie od 0,5 do 6,0 bar.' | JA: 'ワイヤーホルダーの絶縁ジャケットへの印象を避けるために、ワイヤーホルダーの空気圧を0.5〜6 barに設定することができます。' | ZH: '为了避免集线器压触到绝缘皮, 可以把集线器气压调整到0,5到6,0 bar'
  616 = 'Ungarisch' | EN: 'Hungarian' | DE: 'Ungarisch' | FR: 'Hongrois' | HU: 'Magyar' | IT: 'Ungherese' | RU: 'Венге́рский' | RO: 'Maghiară' | ES: 'Húngaro' | PL: 'Węgierski' | JA: 'ハンガリー' | ZH: '匈牙利'
  191 = 'V'
  168 = 'Vorwahl:' | EN: 'Preselection' | DE: 'Vorwahl' | FR: 'Présélection' | HU: 'Eloválasztás' | IT: 'Crimpature impostate' | RU: 'Код' | RO: 'Preselectare' | ES: 'Preselección' | PL: 'Wybór wstępny' | JA: '設定値' | ZH: '预设'
  981 = 'Vorwahl: %d' | EN: 'Preselection: %d' | DE: 'Vorwahl: %d' | FR: 'Présélection: %d' | HU: 'Eloválasztás: %d' | IT: 'Crimpature impostate: %d' | RU: 'Код: %d' | RO: 'Preselectare: %d' | ES: 'Preselección: %d' | PL: 'Wybór wstępny: %d' | JA: '設定値: %d' | ZH: '预设: %d'
  314 = 'Wartungsvorwahl:' | EN: 'Maintenance code' | DE: 'Wartungsvorwahl' | FR: 'Présélection de maintenance' | HU: 'Karbantartás eloválasztása' | IT: 'Manutenzione a (cicli):' | RU: 'Код обслуживания' | RO: 'Codul de intretinere' | ES: 'Código de mantenimiento' | PL: 'Kod obsługi' | JA: 'メンテナンスコード' | ZH: '维护代码'
  188 = 'Wartungszähler:' | EN: 'Maintenance counter' | DE: 'Wartungszähler' | FR: 'Compteur de maintenance' | HU: 'Karbantartás számláló' | IT: 'Contatore totale per manutenzione' | RU: 'Счетчик обслуживания' | RO: 'Numarator intretinere' | ES: 'Contador de mantenimiento' | PL: 'Licznik obsługi' | JA: 'メンテナンスカウンター' | ZH: '保养计数'
  47 = 'Weiter' | EN: 'Next' | DE: 'Weiter'
  934 = 'ZU' | EN: 'CLOSE' | DE: 'ZU'
END_TEXTLIST

// ---- VISUs/Ausstossverz.TcVIS
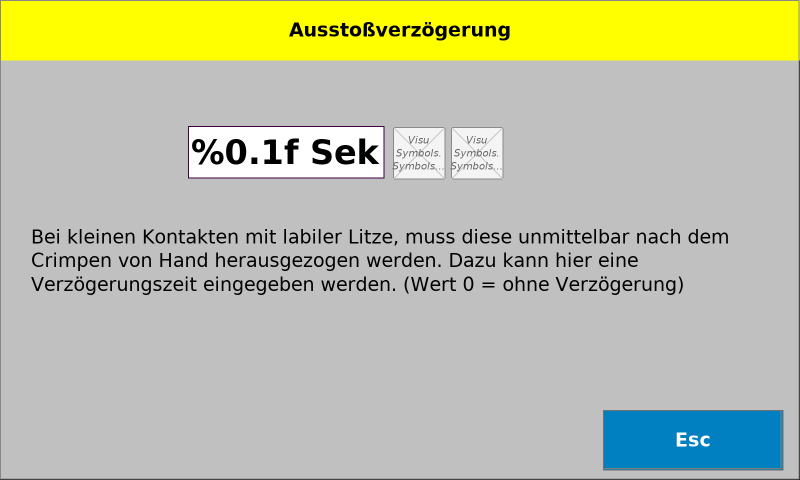
VISUALIZATION Ausstossverz  // 800x480
    Rectangle (0,0 800x480), text variable: DB6.rAusstossverz
    Rectangle (0,0 800x60), "Ausstoßverzögerung"
    Button (603,410 180x60), "Esc"
        OnMouseUp: change screen: Previous 
    Rectangle (188,126 196x52), "%0.1f Sek", text variable: DB6.rAusstossverz
    Image (393,127 52x52), image: VisuSymbols.Symbols.TriangleLeft
        OnMouseClick: execute { P_DecAusstossV(); }
    Image (451,127 52x52), image: VisuSymbols.Symbols.TriangleRight
        OnMouseUp: execute { P_IncAusstossV(); }
    Label (28,224 730x152), "Bei kleinen Kontakten mit labiler Litze, muss diese unmittelbar nach dem Crimpen von Hand herausgezogen werden. Dazu kann hier eine Verzögerungszeit eingegeben werden. (Wert 0 = ohne Verzögerung)"
END_VISUALIZATION

